LIN {X 0,Y 318.181,Z 414.797,A -85,B 0,C 180,E1 -16259.832,E2 -16259.832} C_VEL
LIN {X 0,Y 315.515,Z 502.273,A -85,B 0,C 180,E1 -16261.797,E2 -16261.797} C_VEL
LIN {X 0,Y 314.622,Z 517.231,A -85,B 0,C 180,E1 -16262.298,E2 -16262.298} C_VEL
LIN {X 0,Y 313.283,Z 530.709,A -85,B 0,C 180,E1 -16262.984,E2 -16262.984} C_VEL
LIN {X 0,Y 311.702,Z 543.956,A -85,B 0,C 180,E1 -16263.92,E2 -16263.92} C_VEL
LIN {X 0,Y 309.801,Z 557.279,A -85,B 0,C 180,E1 -16265.151,E2 -16265.151} C_VEL
LIN {X 0,Y 307.763,Z 569.737,A -85,B 0,C 180,E1 -16266.626,E2 -16266.626} C_VEL
LIN {X 0,Y 305.798,Z 579.793,A -85,B 0,C 180,E1 -16268.073,E2 -16268.073} C_VEL
LIN {X 0,Y 303.56,Z 590.854,A -85,B 0,C 180,E1 -16270.035,E2 -16270.035} C_VEL
LIN {X 0,Y 301.653,Z 599.979,A -85,B 0,C 180,E1 -16272.021,E2 -16272.021} C_VEL
LIN {X 0,Y 299.984,Z 608.705,A -85,B 0,C 180,E1 -16274.372,E2 -16274.372} C_VEL
LIN {X 0,Y 298.796,Z 614.845,A -85,B 0,C 180,E1 -16276.398,E2 -16276.398} C_VEL
LIN {X 0,Y 297.807,Z 619.932,A -85,B 0,C 180,E1 -16278.431,E2 -16278.431} C_VEL
LIN {X 0,Y 297.035,Z 625.187,A -85,B 0,C 180,E1 -16281.155,E2 -16281.155} C_VEL
LIN {X 0,Y 296.688,Z 628.133,A -85,B 0,C 180,E1 -16283.2,E2 -16283.2} C_VEL
LIN {X 0,Y 296.486,Z 630.822,A -85,B 0,C 180,E1 -16285.924,E2 -16285.924} C_VEL
LIN {X 0,Y 296.446,Z 632.15,A -85,B 0,C 180,E1 -16288.644,E2 -16288.644} C_VEL
LIN {X 0,Y 296.447,Z 632.143,A -85,B 0,C 180,E1 -16291.36,E2 -16291.36} C_VEL
LIN {X 0,Y 296.487,Z 630.798,A -85,B 0,C 180,E1 -16294.08,E2 -16294.08} C_VEL
LIN {X 0,Y 296.695,Z 628.094,A -85,B 0,C 180,E1 -16296.804,E2 -16296.804} C_VEL
LIN {X 0,Y 297.195,Z 623.958,A -85,B 0,C 180,E1 -16299.53,E2 -16299.53} C_VEL
LIN {X 0,Y 298.059,Z 618.26,A -85,B 0,C 180,E1 -16302.254,E2 -16302.254} C_VEL
LIN {X 0,Y 299.398,Z 611.836,A -85,B 0,C 180,E1 -16304.618,E2 -16304.618} C_VEL
LIN {X 0,Y 300.846,Z 603.858,A -85,B 0,C 180,E1 -16306.98,E2 -16306.98} C_VEL
LIN {X 0,Y 302.56,Z 595.508,A -85,B 0,C 180,E1 -16308.979,E2 -16308.979} C_VEL
LIN {X 0,Y 304.663,Z 585.459,A -85,B 0,C 180,E1 -16310.952,E2 -16310.952} C_VEL
LIN {X 0,Y 306.858,Z 574.243,A -85,B 0,C 180,E1 -16312.738,E2 -16312.738} C_VEL
LIN {X 0,Y 308.806,Z 563.08,A -85,B 0,C 180,E1 -16314.185,E2 -16314.185} C_VEL
LIN {X 0,Y 310.702,Z 550.92,A -85,B 0,C 180,E1 -16315.455,E2 -16315.455} C_VEL
LIN {X 0,Y 312.337,Z 538.56,A -85,B 0,C 180,E1 -16316.477,E2 -16316.477} C_VEL
LIN {X 0,Y 313.896,Z 524.825,A -85,B 0,C 180,E1 -16317.324,E2 -16317.324} C_VEL
LIN {X 0,Y 315.02,Z 510.572,A -85,B 0,C 180,E1 -16317.939,E2 -16317.939} C_VEL
LIN {X 0,Y 315.853,Z 497.641,A -85,B 0,C 180,E1 -16318.356,E2 -16318.356} C_VEL
LIN {X 0,Y 321.075,Z 453.072,A -85,B 0,C 180,E1 -16320.185,E2 -16320.185} C_VEL
LIN {X 0,Y 325.694,Z 416.284,A -85,B 0,C 180,E1 -16321.698,E2 -16321.698} C_VEL
LIN {X 0,Y 325.549,Z 408.176,A -85,B 0,C 180,E1 -16322.367,E2 -16322.367} C_VEL
LIN {X 0,Y 323.178,Z 401.098,A -85,B 0,C 180,E1 -16323.67,E2 -16323.67} C_VEL
LIN {X 0,Y 321.541,Z 396.245,A -85,B 0,C 180,E1 -16324.752,E2 -16324.752} C_VEL
LIN {X 0,Y 321.234,Z 394.789,A -85,B 0,C 180,E1 -16325.171,E2 -16325.171} C_VEL
LIN {X 0,Y 319.761,Z 392.123,A -85,B 0,C 180,E1 -16326.403,E2 -16326.403} C_VEL
LIN {X 0,Y 317.084,Z 387.927,A -85,B 0,C 180,E1 -16329.126,E2 -16329.126} C_VEL
LIN {X 0,Y 315.872,Z 386.212,A -85,B 0,C 180,E1 -16330.845,E2 -16330.845} C_VEL
LIN {X 0,Y 314.928,Z 385.265,A -85,B 0,C 180,E1 -16332.571,E2 -16332.571} C_VEL
LIN {X 0,Y 314.162,Z 384.822,A -85,B 0,C 180,E1 -16335.716,E2 -16335.716} C_VEL
LIN {X 0,Y 314.202,Z 385.504,A -85,B 0,C 180,E1 -16337.853,E2 -16337.853} C_VEL
LIN {X 0,Y 314.421,Z 386.794,A -85,B 0,C 180,E1 -16339.593,E2 -16339.593} C_VEL
LIN {X 0,Y 315.302,Z 390.269,A -85,B 0,C 180,E1 -16342.63,E2 -16342.63} C_VEL
LIN {X 0,Y 318.949,Z 396.314,A -85,B 0,C 180,E1 -16345.133,E2 -16345.133} C_VEL
LIN {X 0,Y 322.085,Z 401.94,A -85,B 0,C 180,E1 -16346.841,E2 -16346.841} C_VEL
LIN {X 0,Y 324.388,Z 406.46,A -85,B 0,C 180,E1 -16347.96,E2 -16347.96} C_VEL
LIN {X 0,Y 327.507,Z 413.311,A -85,B 0,C 180,E1 -16349.361,E2 -16349.361} C_VEL
LIN {X 0,Y 328.621,Z 416.471,A -85,B 0,C 180,E1 -16349.868,E2 -16349.868} C_VEL
LIN {X 0,Y 329.285,Z 421.801,A -85,B 0,C 180,E1 -16350.398,E2 -16350.398} C_VEL
LIN {X 0,Y 320.437,Z 500.804,A -85,B 0,C 180,E1 -16353.544,E2 -16353.544} C_VEL
LIN {X 0,Y 318.54,Z 515.101,A -85,B 0,C 180,E1 -16354.43,E2 -16354.43} C_VEL
LIN {X 0,Y 316.577,Z 526.868,A -85,B 0,C 180,E1 -16355.402,E2 -16355.402} C_VEL
LIN {X 0,Y 314.31,Z 538.512,A -85,B 0,C 180,E1 -16356.616,E2 -16356.616} C_VEL
LIN {X 0,Y 311.806,Z 549.386,A -85,B 0,C 180,E1 -16358.034,E2 -16358.034} C_VEL
LIN {X 0,Y 309.219,Z 559.762,A -85,B 0,C 180,E1 -16359.72,E2 -16359.72} C_VEL
LIN {X 0,Y 306.57,Z 569.095,A -85,B 0,C 180,E1 -16361.626,E2 -16361.626} C_VEL
LIN {X 0,Y 304.38,Z 576.647,A -85,B 0,C 180,E1 -16363.57,E2 -16363.57} C_VEL
LIN {X 0,Y 302.686,Z 581.817,A -85,B 0,C 180,E1 -16365.202,E2 -16365.202} C_VEL
LIN {X 0,Y 301.046,Z 586.845,A -85,B 0,C 180,E1 -16367.186,E2 -16367.186} C_VEL
LIN {X 0,Y 299.652,Z 590.71,A -85,B 0,C 180,E1 -16369.186,E2 -16369.186} C_VEL
LIN {X 0,Y 298.514,Z 593.752,A -85,B 0,C 180,E1 -16371.432,E2 -16371.432} C_VEL
LIN {X 0,Y 297.737,Z 595.31,A -85,B 0,C 180,E1 -16373.222,E2 -16373.222} C_VEL
LIN {X 0,Y 297.348,Z 595.96,A -85,B 0,C 180,E1 -16374.575,E2 -16374.575} C_VEL
LIN {X 0,Y 297.123,Z 596.176,A -85,B 0,C 180,E1 -16375.931,E2 -16375.931} C_VEL
LIN {X 0,Y 296.911,Z 595.987,A -85,B 0,C 180,E1 -16377.287,E2 -16377.287} C_VEL
LIN {X 0,Y 296.735,Z 595.36,A -85,B 0,C 180,E1 -16378.643,E2 -16378.643} C_VEL
LIN {X 0,Y 296.629,Z 594.272,A -85,B 0,C 180,E1 -16380,E2 -16380} C_VEL
LIN {X 0,Y 296.615,Z 592.763,A -85,B 0,C 180,E1 -16381.358,E2 -16381.358} C_VEL
LIN {X 0,Y 296.749,Z 589.624,A -85,B 0,C 180,E1 -16383.394,E2 -16383.394} C_VEL
LIN {X 0,Y 296.833,Z 585.354,A -85,B 0,C 180,E1 -16385.435,E2 -16385.435} C_VEL
LIN {X 0,Y 297.207,Z 578.751,A -85,B 0,C 180,E1 -16387.815,E2 -16387.815} C_VEL
LIN {X 0,Y 297.663,Z 571.555,A -85,B 0,C 180,E1 -16389.856,E2 -16389.856} C_VEL
LIN {X 0,Y 298.297,Z 562.517,A -85,B 0,C 180,E1 -16391.897,E2 -16391.897} C_VEL
LIN {X 0,Y 299.162,Z 552.289,A -85,B 0,C 180,E1 -16393.76,E2 -16393.76} C_VEL
LIN {X 0,Y 300.011,Z 541.96,A -85,B 0,C 180,E1 -16395.28,E2 -16395.28} C_VEL
LIN {X 0,Y 300.804,Z 530.328,A -85,B 0,C 180,E1 -16396.675,E2 -16396.675} C_VEL
LIN {X 0,Y 301.521,Z 518.247,A -85,B 0,C 180,E1 -16397.814,E2 -16397.814} C_VEL
LIN {X 0,Y 302.325,Z 505.7,A -85,B 0,C 180,E1 -16398.729,E2 -16398.729} C_VEL
LIN {X 0,Y 302.867,Z 492.085,A -85,B 0,C 180,E1 -16399.442,E2 -16399.442} C_VEL
LIN {X 0,Y 305.687,Z 408.397,A -85,B 0,C 180,E1 -16402.326,E2 -16402.326} C_VEL
LIN {X 0,Y 302.216,Z 381.764,A -85,B 0,C 180,E1 -16403.423,E2 -16403.423} C_VEL
LIN {X 0,Y 302.408,Z 377.134,A -85,B 0,C 180,E1 -16404.363,E2 -16404.363} C_VEL
LIN {X 0,Y 300.168,Z 364.932,A -85,B 0,C 180,E1 -16407.16,E2 -16407.16} C_VEL
LIN {X 0,Y 298.492,Z 356.928,A -85,B 0,C 180,E1 -16409.062,E2 -16409.062} C_VEL
LIN {X 0,Y 298.403,Z 356.939,A -85,B 0,C 180,E1 -16412.799,E2 -16412.799} C_VEL
LIN {X 0,Y 298.433,Z 356.935,A -85,B 0,C 180,E1 -16416.802,E2 -16416.802} C_VEL
LIN {X 0,Y 298.354,Z 356.945,A -85,B 0,C 180,E1 -16421.267,E2 -16421.267} C_VEL
LIN {X 0,Y 298.361,Z 356.945,A -85,B 0,C 180,E1 -16425.034,E2 -16425.034} C_VEL
LIN {X 0,Y 298.354,Z 356.946,A -85,B 0,C 180,E1 -16428.92,E2 -16428.92} C_VEL
LIN {X 0,Y 298.403,Z 356.941,A -85,B 0,C 180,E1 -16432.238,E2 -16432.238} C_VEL
LIN {X 0,Y 298.498,Z 357.128,A -85,B 0,C 180,E1 -16433.939,E2 -16433.939} C_VEL
LIN {X 0,Y 300.452,Z 364.93,A -85,B 0,C 180,E1 -16436.673,E2 -16436.673} C_VEL
LIN {X 0,Y 309.752,Z 383.967,A -85,B 0,C 180,E1 -16438.311,E2 -16438.311} C_VEL
LIN {X 0,Y 317.575,Z 402.728,A -85,B 0,C 180,E1 -16439.664,E2 -16439.664} C_VEL
LIN {X 0,Y 318.397,Z 408.082,A -85,B 0,C 180,E1 -16439.888,E2 -16439.888} C_VEL
LIN {X 0,Y 315.383,Z 501.879,A -85,B 0,C 180,E1 -16442.006,E2 -16442.006} C_VEL
LIN {X 0,Y 314.601,Z 514.095,A -85,B 0,C 180,E1 -16442.472,E2 -16442.472} C_VEL
LIN {X 0,Y 313.135,Z 528.181,A -85,B 0,C 180,E1 -16443.236,E2 -16443.236} C_VEL
LIN {X 0,Y 311.532,Z 541.631,A -85,B 0,C 180,E1 -16444.259,E2 -16444.259} C_VEL
LIN {X 0,Y 309.826,Z 553.788,A -85,B 0,C 180,E1 -16445.45,E2 -16445.45} C_VEL
LIN {X 0,Y 307.687,Z 566.235,A -85,B 0,C 180,E1 -16446.971,E2 -16446.971} C_VEL
LIN {X 0,Y 305.392,Z 577.917,A -85,B 0,C 180,E1 -16448.747,E2 -16448.747} C_VEL
LIN {X 0,Y 303.28,Z 588.352,A -85,B 0,C 180,E1 -16450.716,E2 -16450.716} C_VEL
LIN {X 0,Y 301.506,Z 596.934,A -85,B 0,C 180,E1 -16452.702,E2 -16452.702} C_VEL
LIN {X 0,Y 299.992,Z 605.205,A -85,B 0,C 180,E1 -16455.064,E2 -16455.064} C_VEL
LIN {X 0,Y 298.702,Z 610.956,A -85,B 0,C 180,E1 -16457.082,E2 -16457.082} C_VEL
LIN {X 0,Y 297.848,Z 615.682,A -85,B 0,C 180,E1 -16459.117,E2 -16459.117} C_VEL
LIN {X 0,Y 297.072,Z 620.571,A -85,B 0,C 180,E1 -16461.838,E2 -16461.838} C_VEL
LIN {X 0,Y 296.69,Z 623.976,A -85,B 0,C 180,E1 -16464.561,E2 -16464.561} C_VEL
LIN {X 0,Y 296.541,Z 626,A -85,B 0,C 180,E1 -16467.281,E2 -16467.281} C_VEL
LIN {X 0,Y 296.452,Z 626.694,A -85,B 0,C 180,E1 -16469.998,E2 -16469.998} C_VEL
LIN {X 0,Y 296.539,Z 626.066,A -85,B 0,C 180,E1 -16472.715,E2 -16472.715} C_VEL
LIN {X 0,Y 296.668,Z 624.104,A -85,B 0,C 180,E1 -16475.435,E2 -16475.435} C_VEL
LIN {X 0,Y 297.056,Z 620.755,A -85,B 0,C 180,E1 -16478.159,E2 -16478.159} C_VEL
LIN {X 0,Y 297.809,Z 615.922,A -85,B 0,C 180,E1 -16480.88,E2 -16480.88} C_VEL
LIN {X 0,Y 299.059,Z 609.457,A -85,B 0,C 180,E1 -16483.59,E2 -16483.59} C_VEL
LIN {X 0,Y 300.295,Z 603.371,A -85,B 0,C 180,E1 -16485.611,E2 -16485.611} C_VEL
LIN {X 0,Y 301.715,Z 596.064,A -85,B 0,C 180,E1 -16487.624,E2 -16487.624} C_VEL
LIN {X 0,Y 303.553,Z 587.276,A -85,B 0,C 180,E1 -16489.613,E2 -16489.613} C_VEL
LIN {X 0,Y 305.738,Z 576.623,A -85,B 0,C 180,E1 -16491.577,E2 -16491.577} C_VEL
LIN {X 0,Y 307.797,Z 565.849,A -85,B 0,C 180,E1 -16493.193,E2 -16493.193} C_VEL
LIN {X 0,Y 309.792,Z 554.196,A -85,B 0,C 180,E1 -16494.617,E2 -16494.617} C_VEL
LIN {X 0,Y 311.623,Z 541.043,A -85,B 0,C 180,E1 -16495.908,E2 -16495.908} C_VEL
LIN {X 0,Y 313.318,Z 527.366,A -85,B 0,C 180,E1 -16496.922,E2 -16496.922} C_VEL
LIN {X 0,Y 314.674,Z 512.864,A -85,B 0,C 180,E1 -16497.697,E2 -16497.697} C_VEL
LIN {X 0,Y 315.593,Z 498.5,A -85,B 0,C 180,E1 -16498.196,E2 -16498.196} C_VEL
LIN {X 0,Y 318.051,Z 420.026,A -85,B 0,C 180,E1 -16499.96,E2 -16499.96} C_VEL
LIN {X 0,Y 317.598,Z 416.226,A -85,B 0,C 180,E1 -16500.104,E2 -16500.104} C_VEL
LIN {X 0,Y 316.27,Z 412.711,A -85,B 0,C 180,E1 -16500.335,E2 -16500.335} C_VEL
LIN {X 0,Y 310.742,Z 402.776,A -85,B 0,C 180,E1 -16501.197,E2 -16501.197} C_VEL
LIN {X 0,Y 310.267,Z 401.571,A -85,B 0,C 180,E1 -16501.282,E2 -16501.282} C_VEL
LIN {X 0,Y 303.441,Z 385.758,A -85,B 0,C 180,E1 -16502.503,E2 -16502.503} C_VEL
LIN {X 0,Y 296.623,Z 371.72,A -85,B 0,C 180,E1 -16503.748,E2 -16503.748} C_VEL
LIN {X 0,Y 293.184,Z 364.851,A -85,B 0,C 180,E1 -16504.427,E2 -16504.427} C_VEL
LIN {X 0,Y 291.391,Z 357.815,A -85,B 0,C 180,E1 -16507.08,E2 -16507.08} C_VEL
LIN {X 0,Y 291.286,Z 357.826,A -85,B 0,C 180,E1 -16511.586,E2 -16511.586} C_VEL
LIN {X 0,Y 291.273,Z 357.827,A -85,B 0,C 180,E1 -16515.594,E2 -16515.594} C_VEL
LIN {X 0,Y 291.29,Z 357.827,A -85,B 0,C 180,E1 -16519.35,E2 -16519.35} C_VEL
LIN {X 0,Y 291.375,Z 357.804,A -85,B 0,C 180,E1 -16522.915,E2 -16522.915} C_VEL
LIN {X 0,Y 291.332,Z 357.807,A -85,B 0,C 180,E1 -16526.3,E2 -16526.3} C_VEL
LIN {X 0,Y 291.352,Z 357.818,A -85,B 0,C 180,E1 -16530.267,E2 -16530.267} C_VEL
LIN {X 0,Y 291.345,Z 357.796,A -85,B 0,C 180,E1 -16534.265,E2 -16534.265} C_VEL
LIN {X 0,Y 291.351,Z 357.817,A -85,B 0,C 180,E1 -16537.297,E2 -16537.297} C_VEL
LIN {X 0,Y 291.379,Z 357.788,A -85,B 0,C 180,E1 -16540.264,E2 -16540.264} C_VEL
LIN {X 0,Y 291.485,Z 357.804,A -85,B 0,C 180,E1 -16544.664,E2 -16544.664} C_VEL
LIN {X 0,Y 291.515,Z 357.799,A -85,B 0,C 180,E1 -16548.88,E2 -16548.88} C_VEL
LIN {X 0,Y 291.636,Z 357.777,A -85,B 0,C 180,E1 -16551.686,E2 -16551.686} C_VEL
LIN {X 0,Y 291.584,Z 357.785,A -85,B 0,C 180,E1 -16554.467,E2 -16554.467} C_VEL
LIN {X 0,Y 291.857,Z 357.752,A -85,B 0,C 180,E1 -16558.62,E2 -16558.62} C_VEL
LIN {X 0,Y 291.866,Z 357.753,A -85,B 0,C 180,E1 -16561.38,E2 -16561.38} C_VEL
LIN {X 0,Y 291.673,Z 357.777,A -85,B 0,C 180,E1 -16566.92,E2 -16566.92} C_VEL
LIN {X 0,Y 291.554,Z 357.789,A -85,B 0,C 180,E1 -16569.714,E2 -16569.714} C_VEL
LIN {X 0,Y 291.501,Z 357.795,A -85,B 0,C 180,E1 -16573.951,E2 -16573.951} C_VEL
LIN {X 0,Y 291.417,Z 357.803,A -85,B 0,C 180,E1 -16576.822,E2 -16576.822} C_VEL
LIN {X 0,Y 291.378,Z 357.812,A -85,B 0,C 180,E1 -16579.843,E2 -16579.843} C_VEL
LIN {X 0,Y 291.313,Z 357.812,A -85,B 0,C 180,E1 -16584.213,E2 -16584.213} C_VEL
LIN {X 0,Y 291.316,Z 357.816,A -85,B 0,C 180,E1 -16587.282,E2 -16587.282} C_VEL
LIN {X 0,Y 291.289,Z 357.815,A -85,B 0,C 180,E1 -16590.442,E2 -16590.442} C_VEL
LIN {X 0,Y 291.332,Z 357.816,A -85,B 0,C 180,E1 -16593.7,E2 -16593.7} C_VEL
LIN {X 0,Y 291.341,Z 357.82,A -85,B 0,C 180,E1 -16597.249,E2 -16597.249} C_VEL
LIN {X 0,Y 291.288,Z 357.824,A -85,B 0,C 180,E1 -16600.65,E2 -16600.65} C_VEL
LIN {X 0,Y 291.272,Z 357.831,A -85,B 0,C 180,E1 -16604.405,E2 -16604.405} C_VEL
LIN {X 0,Y 291.285,Z 357.83,A -85,B 0,C 180,E1 -16608.413,E2 -16608.413} C_VEL
LIN {X 0,Y 291.364,Z 357.957,A -85,B 0,C 180,E1 -16611.73,E2 -16611.73} C_VEL
LIN {X 0,Y 293.787,Z 366.948,A -85,B 0,C 180,E1 -16614.964,E2 -16614.964} C_VEL
LIN {X 0,Y 294.381,Z 369.415,A -85,B 0,C 180,E1 -16615.805,E2 -16615.805} C_VEL
LIN {X 0,Y 303.664,Z 388.91,A -85,B 0,C 180,E1 -16617.522,E2 -16617.522} C_VEL
LIN {X 0,Y 309.907,Z 403.802,A -85,B 0,C 180,E1 -16618.649,E2 -16618.649} C_VEL
LIN {X 0,Y 312.081,Z 416.22,A -85,B 0,C 180,E1 -16619.217,E2 -16619.217} C_VEL
LIN {X 0,Y 309.113,Z 506.688,A -85,B 0,C 180,E1 -16621.298,E2 -16621.298} C_VEL
LIN {X 0,Y 308.029,Z 520.691,A -85,B 0,C 180,E1 -16621.838,E2 -16621.838} C_VEL
LIN {X 0,Y 306.571,Z 534.345,A -85,B 0,C 180,E1 -16622.62,E2 -16622.62} C_VEL
LIN {X 0,Y 304.792,Z 547.616,A -85,B 0,C 180,E1 -16623.651,E2 -16623.651} C_VEL
LIN {X 0,Y 302.863,Z 560.156,A -85,B 0,C 180,E1 -16624.916,E2 -16624.916} C_VEL
LIN {X 0,Y 300.81,Z 572.022,A -85,B 0,C 180,E1 -16626.418,E2 -16626.418} C_VEL
LIN {X 0,Y 298.742,Z 581.694,A -85,B 0,C 180,E1 -16627.891,E2 -16627.891} C_VEL
LIN {X 0,Y 296.499,Z 592.417,A -85,B 0,C 180,E1 -16629.9,E2 -16629.9} C_VEL
LIN {X 0,Y 294.563,Z 601.27,A -85,B 0,C 180,E1 -16631.933,E2 -16631.933} C_VEL
LIN {X 0,Y 292.871,Z 609.756,A -85,B 0,C 180,E1 -16634.34,E2 -16634.34} C_VEL
LIN {X 0,Y 291.477,Z 616.591,A -85,B 0,C 180,E1 -16636.761,E2 -16636.761} C_VEL
LIN {X 0,Y 290.577,Z 621.302,A -85,B 0,C 180,E1 -16638.846,E2 -16638.846} C_VEL
LIN {X 0,Y 289.846,Z 626.189,A -85,B 0,C 180,E1 -16641.637,E2 -16641.637} C_VEL
LIN {X 0,Y 289.471,Z 629.68,A -85,B 0,C 180,E1 -16644.521,E2 -16644.521} C_VEL
LIN {X 0,Y 289.388,Z 631.588,A -85,B 0,C 180,E1 -16647.218,E2 -16647.218} C_VEL
LIN {X 0,Y 289.37,Z 632.246,A -85,B 0,C 180,E1 -16650.002,E2 -16650.002} C_VEL
LIN {X 0,Y 289.389,Z 631.571,A -85,B 0,C 180,E1 -16652.786,E2 -16652.786} C_VEL
LIN {X 0,Y 289.481,Z 629.551,A -85,B 0,C 180,E1 -16655.575,E2 -16655.575} C_VEL
LIN {X 0,Y 289.861,Z 626.143,A -85,B 0,C 180,E1 -16658.367,E2 -16658.367} C_VEL
LIN {X 0,Y 290.58,Z 621.246,A -85,B 0,C 180,E1 -16661.158,E2 -16661.158} C_VEL
LIN {X 0,Y 291.481,Z 616.519,A -85,B 0,C 180,E1 -16663.244,E2 -16663.244} C_VEL
LIN {X 0,Y 292.868,Z 609.664,A -85,B 0,C 180,E1 -16665.664,E2 -16665.664} C_VEL
LIN {X 0,Y 294.566,Z 601.158,A -85,B 0,C 180,E1 -16668.071,E2 -16668.071} C_VEL
LIN {X 0,Y 296.502,Z 592.281,A -85,B 0,C 180,E1 -16670.104,E2 -16670.104} C_VEL
LIN {X 0,Y 298.747,Z 581.531,A -85,B 0,C 180,E1 -16672.113,E2 -16672.113} C_VEL
LIN {X 0,Y 300.989,Z 570.65,A -85,B 0,C 180,E1 -16673.754,E2 -16673.754} C_VEL
LIN {X 0,Y 303.132,Z 558.555,A -85,B 0,C 180,E1 -16675.241,E2 -16675.241} C_VEL
LIN {X 0,Y 305.032,Z 545.501,A -85,B 0,C 180,E1 -16676.515,E2 -16676.515} C_VEL
LIN {X 0,Y 307.888,Z 525.854,A -85,B 0,C 180,E1 -16677.995,E2 -16677.995} C_VEL
LIN {X 0,Y 309.583,Z 512.084,A -85,B 0,C 180,E1 -16678.752,E2 -16678.752} C_VEL
LIN {X 0,Y 316.684,Z 455.092,A -85,B 0,C 180,E1 -16681.141,E2 -16681.141} C_VEL
LIN {X 0,Y 321.69,Z 418.334,A -85,B 0,C 180,E1 -16682.669,E2 -16682.669} C_VEL
LIN {X 0,Y 321.657,Z 412.005,A -85,B 0,C 180,E1 -16683.213,E2 -16683.213} C_VEL
LIN {X 0,Y 319.912,Z 406.208,A -85,B 0,C 180,E1 -16684.323,E2 -16684.323} C_VEL
LIN {X 0,Y 317.902,Z 400.512,A -85,B 0,C 180,E1 -16685.657,E2 -16685.657} C_VEL
LIN {X 0,Y 314.755,Z 396.173,A -85,B 0,C 180,E1 -16687.662,E2 -16687.662} C_VEL
LIN {X 0,Y 313.481,Z 394.308,A -85,B 0,C 180,E1 -16688.885,E2 -16688.885} C_VEL
LIN {X 0,Y 312.065,Z 392.237,A -85,B 0,C 180,E1 -16690.778,E2 -16690.778} C_VEL
LIN {X 0,Y 310.582,Z 390.824,A -85,B 0,C 180,E1 -16693.605,E2 -16693.605} C_VEL
LIN {X 0,Y 310.017,Z 390.757,A -85,B 0,C 180,E1 -16696.507,E2 -16696.507} C_VEL
LIN {X 0,Y 310.122,Z 392.046,A -85,B 0,C 180,E1 -16698.913,E2 -16698.913} C_VEL
LIN {X 0,Y 312.611,Z 396.096,A -85,B 0,C 180,E1 -16701.895,E2 -16701.895} C_VEL
LIN {X 0,Y 315.852,Z 401.54,A -85,B 0,C 180,E1 -16704.393,E2 -16704.393} C_VEL
LIN {X 0,Y 318.844,Z 407.285,A -85,B 0,C 180,E1 -16706.215,E2 -16706.215} C_VEL
LIN {X 0,Y 321.387,Z 412.56,A -85,B 0,C 180,E1 -16707.564,E2 -16707.564} C_VEL
LIN {X 0,Y 324.493,Z 419.929,A -85,B 0,C 180,E1 -16709.054,E2 -16709.054} C_VEL
LIN {X 0,Y 324.888,Z 423.919,A -85,B 0,C 180,E1 -16709.461,E2 -16709.461} C_VEL
LIN {X 0,Y 315.587,Z 501.078,A -85,B 0,C 180,E1 -16712.612,E2 -16712.612} C_VEL
LIN {X 0,Y 313.452,Z 515.756,A -85,B 0,C 180,E1 -16713.537,E2 -16713.537} C_VEL
LIN {X 0,Y 311.208,Z 528.176,A -85,B 0,C 180,E1 -16714.591,E2 -16714.591} C_VEL
LIN {X 0,Y 308.499,Z 540.821,A -85,B 0,C 180,E1 -16715.97,E2 -16715.97} C_VEL
LIN {X 0,Y 305.659,Z 552.109,A -85,B 0,C 180,E1 -16717.526,E2 -16717.526} C_VEL
LIN {X 0,Y 302.852,Z 562.164,A -85,B 0,C 180,E1 -16719.275,E2 -16719.275} C_VEL
LIN {X 0,Y 300.086,Z 571.129,A -85,B 0,C 180,E1 -16721.215,E2 -16721.215} C_VEL
LIN {X 0,Y 297.374,Z 579.378,A -85,B 0,C 180,E1 -16723.525,E2 -16723.525} C_VEL
LIN {X 0,Y 295.382,Z 584.987,A -85,B 0,C 180,E1 -16725.533,E2 -16725.533} C_VEL
LIN {X 0,Y 293.64,Z 589.407,A -85,B 0,C 180,E1 -16727.561,E2 -16727.561} C_VEL
LIN {X 0,Y 292.753,Z 591.686,A -85,B 0,C 180,E1 -16728.927,E2 -16728.927} C_VEL
LIN {X 0,Y 291.484,Z 594.625,A -85,B 0,C 180,E1 -16731.332,E2 -16731.332} C_VEL
LIN {X 0,Y 290.734,Z 595.92,A -85,B 0,C 180,E1 -16733.058,E2 -16733.058} C_VEL
LIN {X 0,Y 290.311,Z 596.458,A -85,B 0,C 180,E1 -16734.443,E2 -16734.443} C_VEL
LIN {X 0,Y 290.056,Z 596.585,A -85,B 0,C 180,E1 -16735.832,E2 -16735.832} C_VEL
LIN {X 0,Y 289.832,Z 596.275,A -85,B 0,C 180,E1 -16737.22,E2 -16737.22} C_VEL
LIN {X 0,Y 289.65,Z 595.513,A -85,B 0,C 180,E1 -16738.61,E2 -16738.61} C_VEL
LIN {X 0,Y 289.543,Z 594.338,A -85,B 0,C 180,E1 -16740,E2 -16740} C_VEL
LIN {X 0,Y 289.553,Z 591.724,A -85,B 0,C 180,E1 -16742.087,E2 -16742.087} C_VEL
LIN {X 0,Y 289.698,Z 588.036,A -85,B 0,C 180,E1 -16744.174,E2 -16744.174} C_VEL
LIN {X 0,Y 289.894,Z 582.403,A -85,B 0,C 180,E1 -16746.542,E2 -16746.542} C_VEL
LIN {X 0,Y 290.264,Z 575.769,A -85,B 0,C 180,E1 -16748.704,E2 -16748.704} C_VEL
LIN {X 0,Y 290.836,Z 567.725,A -85,B 0,C 180,E1 -16750.794,E2 -16750.794} C_VEL
LIN {X 0,Y 291.601,Z 557.661,A -85,B 0,C 180,E1 -16752.882,E2 -16752.882} C_VEL
LIN {X 0,Y 292.369,Z 548.439,A -85,B 0,C 180,E1 -16754.442,E2 -16754.442} C_VEL
LIN {X 0,Y 293.255,Z 537.159,A -85,B 0,C 180,E1 -16755.998,E2 -16755.998} C_VEL
LIN {X 0,Y 294.14,Z 524.634,A -85,B 0,C 180,E1 -16757.377,E2 -16757.377} C_VEL
LIN {X 0,Y 294.943,Z 511.46,A -85,B 0,C 180,E1 -16758.495,E2 -16758.495} C_VEL
LIN {X 0,Y 295.618,Z 497.641,A -85,B 0,C 180,E1 -16759.351,E2 -16759.351} C_VEL
LIN {X 0,Y 296.256,Z 482.294,A -85,B 0,C 180,E1 -16759.984,E2 -16759.984} C_VEL
LIN {X 0,Y 298.73,Z 409.096,A -85,B 0,C 180,E1 -16762.579,E2 -16762.579} C_VEL
LIN {X 0,Y 295.229,Z 381.64,A -85,B 0,C 180,E1 -16763.758,E2 -16763.758} C_VEL
LIN {X 0,Y 295.389,Z 377.94,A -85,B 0,C 180,E1 -16764.56,E2 -16764.56} C_VEL
LIN {X 0,Y 292.812,Z 364.332,A -85,B 0,C 180,E1 -16767.729,E2 -16767.729} C_VEL
LIN {X 0,Y 291.455,Z 357.805,A -85,B 0,C 180,E1 -16769.286,E2 -16769.286} C_VEL
LIN {X 0,Y 291.352,Z 357.816,A -85,B 0,C 180,E1 -16773.698,E2 -16773.698} C_VEL
LIN {X 0,Y 291.359,Z 357.817,A -85,B 0,C 180,E1 -16777.247,E2 -16777.247} C_VEL
LIN {X 0,Y 291.301,Z 357.825,A -85,B 0,C 180,E1 -16781.588,E2 -16781.588} C_VEL
LIN {X 0,Y 291.288,Z 357.828,A -85,B 0,C 180,E1 -16785.595,E2 -16785.595} C_VEL
LIN {X 0,Y 291.306,Z 357.826,A -85,B 0,C 180,E1 -16789.351,E2 -16789.351} C_VEL
LIN {X 0,Y 291.408,Z 357.852,A -85,B 0,C 180,E1 -16793.134,E2 -16793.134} C_VEL
LIN {X 0,Y 293.312,Z 365.196,A -85,B 0,C 180,E1 -16795.755,E2 -16795.755} C_VEL
LIN {X 0,Y 302.995,Z 384.698,A -85,B 0,C 180,E1 -16797.536,E2 -16797.536} C_VEL
LIN {X 0,Y 310.198,Z 401.425,A -85,B 0,C 180,E1 -16798.826,E2 -16798.826} C_VEL
LIN {X 0,Y 311.886,Z 406.121,A -85,B 0,C 180,E1 -16799.138,E2 -16799.138} C_VEL
LIN {X 0,Y 312.27,Z 408.498,A -85,B 0,C 180,E1 -16799.242,E2 -16799.242} C_VEL
LIN {X 0,Y 309.149,Z 501.962,A -85,B 0,C 180,E1 -16801.39,E2 -16801.39} C_VEL
LIN {X 0,Y 308.315,Z 514.175,A -85,B 0,C 180,E1 -16801.862,E2 -16801.862} C_VEL
LIN {X 0,Y 306.818,Z 528.256,A -85,B 0,C 180,E1 -16802.64,E2 -16802.64} C_VEL
LIN {X 0,Y 305.15,Z 541.704,A -85,B 0,C 180,E1 -16803.68,E2 -16803.68} C_VEL
LIN {X 0,Y 303.309,Z 554.271,A -85,B 0,C 180,E1 -16804.939,E2 -16804.939} C_VEL
LIN {X 0,Y 301.154,Z 566.307,A -85,B 0,C 180,E1 -16806.442,E2 -16806.442} C_VEL
LIN {X 0,Y 298.769,Z 577.988,A -85,B 0,C 180,E1 -16808.252,E2 -16808.252} C_VEL
LIN {X 0,Y 296.576,Z 588.423,A -85,B 0,C 180,E1 -16810.262,E2 -16810.262} C_VEL
LIN {X 0,Y 294.642,Z 597.296,A -85,B 0,C 180,E1 -16812.364,E2 -16812.364} C_VEL
LIN {X 0,Y 293.101,Z 605.274,A -85,B 0,C 180,E1 -16814.705,E2 -16814.705} C_VEL
LIN {X 0,Y 291.75,Z 611.026,A -85,B 0,C 180,E1 -16816.769,E2 -16816.769} C_VEL
LIN {X 0,Y 290.843,Z 615.751,A -85,B 0,C 180,E1 -16818.852,E2 -16818.852} C_VEL
LIN {X 0,Y 290.019,Z 620.64,A -85,B 0,C 180,E1 -16821.638,E2 -16821.638} C_VEL
LIN {X 0,Y 289.606,Z 624.044,A -85,B 0,C 180,E1 -16824.428,E2 -16824.428} C_VEL
LIN {X 0,Y 289.448,Z 626.067,A -85,B 0,C 180,E1 -16827.214,E2 -16827.214} C_VEL
LIN {X 0,Y 289.373,Z 626.761,A -85,B 0,C 180,E1 -16829.998,E2 -16829.998} C_VEL
LIN {X 0,Y 289.446,Z 626.133,A -85,B 0,C 180,E1 -16832.781,E2 -16832.781} C_VEL
LIN {X 0,Y 289.604,Z 624.17,A -85,B 0,C 180,E1 -16835.568,E2 -16835.568} C_VEL
LIN {X 0,Y 290.007,Z 620.822,A -85,B 0,C 180,E1 -16838.358,E2 -16838.358} C_VEL
LIN {X 0,Y 290.81,Z 615.988,A -85,B 0,C 180,E1 -16841.145,E2 -16841.145} C_VEL
LIN {X 0,Y 291.722,Z 611.327,A -85,B 0,C 180,E1 -16843.228,E2 -16843.228} C_VEL
LIN {X 0,Y 293.243,Z 604.55,A -85,B 0,C 180,E1 -16845.639,E2 -16845.639} C_VEL
LIN {X 0,Y 294.636,Z 597.524,A -85,B 0,C 180,E1 -16847.691,E2 -16847.691} C_VEL
LIN {X 0,Y 296.507,Z 588.96,A -85,B 0,C 180,E1 -16849.738,E2 -16849.738} C_VEL
LIN {X 0,Y 298.732,Z 578.635,A -85,B 0,C 180,E1 -16851.746,E2 -16851.746} C_VEL
LIN {X 0,Y 301.047,Z 567.084,A -85,B 0,C 180,E1 -16853.562,E2 -16853.562} C_VEL
LIN {X 0,Y 303.129,Z 555.768,A -85,B 0,C 180,E1 -16855.001,E2 -16855.001} C_VEL
LIN {X 0,Y 304.782,Z 544.635,A -85,B 0,C 180,E1 -16856.166,E2 -16856.166} C_VEL
LIN {X 0,Y 306.453,Z 531.993,A -85,B 0,C 180,E1 -16857.206,E2 -16857.206} C_VEL
LIN {X 0,Y 307.963,Z 517.806,A -85,B 0,C 180,E1 -16858.076,E2 -16858.076} C_VEL
LIN {X 0,Y 309.064,Z 503.825,A -85,B 0,C 180,E1 -16858.661,E2 -16858.661} C_VEL
LIN {X 0,Y 310.047,Z 479.535,A -85,B 0,C 180,E1 -16859.257,E2 -16859.257} C_VEL
LIN {X 0,Y 312.254,Z 407.787,A -85,B 0,C 180,E1 -16860.897,E2 -16860.897} C_VEL
LIN {X 0,Y 311.265,Z 404.16,A -85,B 0,C 180,E1 -16861.102,E2 -16861.102} C_VEL
LIN {X 0,Y 310.267,Z 401.571,A -85,B 0,C 180,E1 -16861.282,E2 -16861.282} C_VEL
LIN {X 0,Y 307.751,Z 396.737,A -85,B 0,C 180,E1 -16861.697,E2 -16861.697} C_VEL
LIN {X 0,Y 304.401,Z 392.617,A -85,B 0,C 180,E1 -16862.2,E2 -16862.2} C_VEL
LIN {X 0,Y 295.996,Z 383.65,A -85,B 0,C 180,E1 -16863.488,E2 -16863.488} C_VEL
LIN {X 0,Y 293.178,Z 379.055,A -85,B 0,C 180,E1 -16863.987,E2 -16863.987} C_VEL
LIN {X 0,Y 285.997,Z 364.972,A -85,B 0,C 180,E1 -16865.406,E2 -16865.406} C_VEL
LIN {X 0,Y 284.29,Z 358.698,A -85,B 0,C 180,E1 -16867.879,E2 -16867.879} C_VEL
LIN {X 0,Y 284.228,Z 358.704,A -85,B 0,C 180,E1 -16872.115,E2 -16872.115} C_VEL
LIN {X 0,Y 284.229,Z 358.704,A -85,B 0,C 180,E1 -16876.184,E2 -16876.184} C_VEL
LIN {X 0,Y 284.273,Z 358.7,A -85,B 0,C 180,E1 -16880.028,E2 -16880.028} C_VEL
LIN {X 0,Y 284.308,Z 358.692,A -85,B 0,C 180,E1 -16883.61,E2 -16883.61} C_VEL
LIN {X 0,Y 284.295,Z 358.677,A -85,B 0,C 180,E1 -16887.189,E2 -16887.189} C_VEL
LIN {X 0,Y 284.324,Z 358.694,A -85,B 0,C 180,E1 -16890.372,E2 -16890.372} C_VEL
LIN {X 0,Y 284.292,Z 358.671,A -85,B 0,C 180,E1 -16893.578,E2 -16893.578} C_VEL
LIN {X 0,Y 284.314,Z 358.695,A -85,B 0,C 180,E1 -16896.702,E2 -16896.702} C_VEL
LIN {X 0,Y 284.319,Z 358.666,A -85,B 0,C 180,E1 -16901.256,E2 -16901.256} C_VEL
LIN {X 0,Y 284.449,Z 358.675,A -85,B 0,C 180,E1 -16905.695,E2 -16905.695} C_VEL
LIN {X 0,Y 284.5,Z 358.669,A -85,B 0,C 180,E1 -16910.042,E2 -16910.042} C_VEL
LIN {X 0,Y 284.626,Z 358.657,A -85,B 0,C 180,E1 -16912.908,E2 -16912.908} C_VEL
LIN {X 0,Y 284.824,Z 358.628,A -85,B 0,C 180,E1 -16918.586,E2 -16918.586} C_VEL
LIN {X 0,Y 284.832,Z 358.629,A -85,B 0,C 180,E1 -16921.414,E2 -16921.414} C_VEL
LIN {X 0,Y 284.628,Z 358.653,A -85,B 0,C 180,E1 -16927.092,E2 -16927.092} C_VEL
LIN {X 0,Y 284.5,Z 358.669,A -85,B 0,C 180,E1 -16929.958,E2 -16929.958} C_VEL
LIN {X 0,Y 284.449,Z 358.676,A -85,B 0,C 180,E1 -16934.304,E2 -16934.304} C_VEL
LIN {X 0,Y 284.32,Z 358.694,A -85,B 0,C 180,E1 -16938.744,E2 -16938.744} C_VEL
LIN {X 0,Y 284.294,Z 358.676,A -85,B 0,C 180,E1 -16943.299,E2 -16943.299} C_VEL
LIN {X 0,Y 284.273,Z 358.694,A -85,B 0,C 180,E1 -16947.131,E2 -16947.131} C_VEL
LIN {X 0,Y 284.261,Z 358.687,A -85,B 0,C 180,E1 -16950.085,E2 -16950.085} C_VEL
LIN {X 0,Y 284.293,Z 358.693,A -85,B 0,C 180,E1 -16952.947,E2 -16952.947} C_VEL
LIN {X 0,Y 284.306,Z 358.694,A -85,B 0,C 180,E1 -16956.39,E2 -16956.39} C_VEL
LIN {X 0,Y 284.271,Z 358.702,A -85,B 0,C 180,E1 -16960.001,E2 -16960.001} C_VEL
LIN {X 0,Y 284.223,Z 358.707,A -85,B 0,C 180,E1 -16964.19,E2 -16964.19} C_VEL
LIN {X 0,Y 284.23,Z 358.709,A -85,B 0,C 180,E1 -16968.12,E2 -16968.12} C_VEL
LIN {X 0,Y 284.327,Z 358.839,A -85,B 0,C 180,E1 -16970.93,E2 -16970.93} C_VEL
LIN {X 0,Y 286.797,Z 368.082,A -85,B 0,C 180,E1 -16974.373,E2 -16974.373} C_VEL
LIN {X 0,Y 287.223,Z 369.574,A -85,B 0,C 180,E1 -16974.836,E2 -16974.836} C_VEL
LIN {X 0,Y 296.596,Z 388.69,A -85,B 0,C 180,E1 -16976.644,E2 -16976.644} C_VEL
LIN {X 0,Y 303.957,Z 405.993,A -85,B 0,C 180,E1 -16978.024,E2 -16978.024} C_VEL
LIN {X 0,Y 305.958,Z 417.321,A -85,B 0,C 180,E1 -16978.563,E2 -16978.563} C_VEL
LIN {X 0,Y 302.913,Z 506.636,A -85,B 0,C 180,E1 -16980.654,E2 -16980.654} C_VEL
LIN {X 0,Y 301.771,Z 520.632,A -85,B 0,C 180,E1 -16981.2,E2 -16981.2} C_VEL
LIN {X 0,Y 300.284,Z 534.284,A -85,B 0,C 180,E1 -16981.997,E2 -16981.997} C_VEL
LIN {X 0,Y 298.429,Z 547.554,A -85,B 0,C 180,E1 -16983.045,E2 -16983.045} C_VEL
LIN {X 0,Y 296.274,Z 560.983,A -85,B 0,C 180,E1 -16984.435,E2 -16984.435} C_VEL
LIN {X 0,Y 294.049,Z 573.132,A -85,B 0,C 180,E1 -16986.029,E2 -16986.029} C_VEL
LIN {X 0,Y 291.73,Z 583.583,A -85,B 0,C 180,E1 -16987.704,E2 -16987.704} C_VEL
LIN {X 0,Y 289.47,Z 593.981,A -85,B 0,C 180,E1 -16989.761,E2 -16989.761} C_VEL
LIN {X 0,Y 287.475,Z 602.56,A -85,B 0,C 180,E1 -16991.841,E2 -16991.841} C_VEL
LIN {X 0,Y 285.754,Z 610.774,A -85,B 0,C 180,E1 -16994.306,E2 -16994.306} C_VEL
LIN {X 0,Y 284.549,Z 616.525,A -85,B 0,C 180,E1 -16996.432,E2 -16996.432} C_VEL
LIN {X 0,Y 283.554,Z 621.235,A -85,B 0,C 180,E1 -16998.566,E2 -16998.566} C_VEL
LIN {X 0,Y 282.792,Z 626.122,A -85,B 0,C 180,E1 -17001.427,E2 -17001.427} C_VEL
LIN {X 0,Y 282.385,Z 629.517,A -85,B 0,C 180,E1 -17004.289,E2 -17004.289} C_VEL
LIN {X 0,Y 282.298,Z 631.521,A -85,B 0,C 180,E1 -17007.148,E2 -17007.148} C_VEL
LIN {X 0,Y 282.293,Z 632.179,A -85,B 0,C 180,E1 -17010.002,E2 -17010.002} C_VEL
LIN {X 0,Y 282.298,Z 631.503,A -85,B 0,C 180,E1 -17012.856,E2 -17012.856} C_VEL
LIN {X 0,Y 282.408,Z 629.483,A -85,B 0,C 180,E1 -17015.715,E2 -17015.715} C_VEL
LIN {X 0,Y 282.803,Z 626.075,A -85,B 0,C 180,E1 -17018.577,E2 -17018.577} C_VEL
LIN {X 0,Y 283.558,Z 621.177,A -85,B 0,C 180,E1 -17021.438,E2 -17021.438} C_VEL
LIN {X 0,Y 284.552,Z 616.45,A -85,B 0,C 180,E1 -17023.572,E2 -17023.572} C_VEL
LIN {X 0,Y 285.989,Z 609.685,A -85,B 0,C 180,E1 -17026.022,E2 -17026.022} C_VEL
LIN {X 0,Y 287.483,Z 602.444,A -85,B 0,C 180,E1 -17028.163,E2 -17028.163} C_VEL
LIN {X 0,Y 289.471,Z 593.841,A -85,B 0,C 180,E1 -17030.243,E2 -17030.243} C_VEL
LIN {X 0,Y 291.735,Z 583.413,A -85,B 0,C 180,E1 -17032.3,E2 -17032.3} C_VEL
LIN {X 0,Y 294.26,Z 571.784,A -85,B 0,C 180,E1 -17034.144,E2 -17034.144} C_VEL
LIN {X 0,Y 298.107,Z 552.979,A -85,B 0,C 180,E1 -17036.613,E2 -17036.613} C_VEL
LIN {X 0,Y 300.311,Z 542.26,A -85,B 0,C 180,E1 -17037.72,E2 -17037.72} C_VEL
LIN {X 0,Y 302.877,Z 527.859,A -85,B 0,C 180,E1 -17038.879,E2 -17038.879} C_VEL
LIN {X 0,Y 304.891,Z 513.756,A -85,B 0,C 180,E1 -17039.711,E2 -17039.711} C_VEL
LIN {X 0,Y 312.719,Z 455.538,A -85,B 0,C 180,E1 -17042.214,E2 -17042.214} C_VEL
LIN {X 0,Y 317.922,Z 419.724,A -85,B 0,C 180,E1 -17043.738,E2 -17043.738} C_VEL
LIN {X 0,Y 317.952,Z 415.898,A -85,B 0,C 180,E1 -17044.083,E2 -17044.083} C_VEL
LIN {X 0,Y 316.446,Z 410.532,A -85,B 0,C 180,E1 -17045.175,E2 -17045.175} C_VEL
LIN {X 0,Y 315.104,Z 406.404,A -85,B 0,C 180,E1 -17046.192,E2 -17046.192} C_VEL
LIN {X 0,Y 312.295,Z 402.41,A -85,B 0,C 180,E1 -17048.128,E2 -17048.128} C_VEL
LIN {X 0,Y 309.777,Z 399.218,A -85,B 0,C 180,E1 -17050.444,E2 -17050.444} C_VEL
LIN {X 0,Y 308.215,Z 397.691,A -85,B 0,C 180,E1 -17052.611,E2 -17052.611} C_VEL
LIN {X 0,Y 307.427,Z 397.195,A -85,B 0,C 180,E1 -17055.13,E2 -17055.13} C_VEL
LIN {X 0,Y 307.754,Z 397.917,A -85,B 0,C 180,E1 -17057.531,E2 -17057.531} C_VEL
LIN {X 0,Y 308.659,Z 399.579,A -85,B 0,C 180,E1 -17059.415,E2 -17059.415} C_VEL
LIN {X 0,Y 311.016,Z 403.602,A -85,B 0,C 180,E1 -17062.119,E2 -17062.119} C_VEL
LIN {X 0,Y 313.822,Z 408.862,A -85,B 0,C 180,E1 -17064.351,E2 -17064.351} C_VEL
LIN {X 0,Y 316.37,Z 414.034,A -85,B 0,C 180,E1 -17065.973,E2 -17065.973} C_VEL
LIN {X 0,Y 318.984,Z 420.011,A -85,B 0,C 180,E1 -17067.447,E2 -17067.447} C_VEL
LIN {X 0,Y 320.653,Z 424.564,A -85,B 0,C 180,E1 -17068.344,E2 -17068.344} C_VEL
LIN {X 0,Y 320.633,Z 426.569,A -85,B 0,C 180,E1 -17068.504,E2 -17068.504} C_VEL
LIN {X 0,Y 310.865,Z 501.845,A -85,B 0,C 180,E1 -17071.656,E2 -17071.656} C_VEL
LIN {X 0,Y 308.673,Z 515.78,A -85,B 0,C 180,E1 -17072.544,E2 -17072.544} C_VEL
LIN {X 0,Y 306.275,Z 528.178,A -85,B 0,C 180,E1 -17073.602,E2 -17073.602} C_VEL
LIN {X 0,Y 303.459,Z 540.564,A -85,B 0,C 180,E1 -17074.961,E2 -17074.961} C_VEL
LIN {X 0,Y 300.338,Z 552.106,A -85,B 0,C 180,E1 -17076.559,E2 -17076.559} C_VEL
LIN {X 0,Y 297.576,Z 561.391,A -85,B 0,C 180,E1 -17078.163,E2 -17078.163} C_VEL
LIN {X 0,Y 294.584,Z 570.483,A -85,B 0,C 180,E1 -17080.125,E2 -17080.125} C_VEL
LIN {X 0,Y 292.361,Z 576.741,A -85,B 0,C 180,E1 -17081.79,E2 -17081.79} C_VEL
LIN {X 0,Y 290.005,Z 582.96,A -85,B 0,C 180,E1 -17083.818,E2 -17083.818} C_VEL
LIN {X 0,Y 288.045,Z 587.887,A -85,B 0,C 180,E1 -17085.878,E2 -17085.878} C_VEL
LIN {X 0,Y 286.279,Z 591.688,A -85,B 0,C 180,E1 -17087.956,E2 -17087.956} C_VEL
LIN {X 0,Y 285.146,Z 594.405,A -85,B 0,C 180,E1 -17090.065,E2 -17090.065} C_VEL
LIN {X 0,Y 284.36,Z 595.67,A -85,B 0,C 180,E1 -17091.472,E2 -17091.472} C_VEL
LIN {X 0,Y 283.735,Z 596.521,A -85,B 0,C 180,E1 -17092.886,E2 -17092.886} C_VEL
LIN {X 0,Y 283.277,Z 596.963,A -85,B 0,C 180,E1 -17094.305,E2 -17094.305} C_VEL
LIN {X 0,Y 282.994,Z 596.952,A -85,B 0,C 180,E1 -17095.727,E2 -17095.727} C_VEL
LIN {X 0,Y 282.756,Z 596.506,A -85,B 0,C 180,E1 -17097.151,E2 -17097.151} C_VEL
LIN {X 0,Y 282.567,Z 595.653,A -85,B 0,C 180,E1 -17098.575,E2 -17098.575} C_VEL
LIN {X 0,Y 282.458,Z 594.367,A -85,B 0,C 180,E1 -17100,E2 -17100} C_VEL
LIN {X 0,Y 282.479,Z 591.568,A -85,B 0,C 180,E1 -17102.139,E2 -17102.139} C_VEL
LIN {X 0,Y 282.617,Z 587.678,A -85,B 0,C 180,E1 -17104.279,E2 -17104.279} C_VEL
LIN {X 0,Y 282.787,Z 582.585,A -85,B 0,C 180,E1 -17106.421,E2 -17106.421} C_VEL
LIN {X 0,Y 283.153,Z 576.134,A -85,B 0,C 180,E1 -17108.565,E2 -17108.565} C_VEL
LIN {X 0,Y 283.692,Z 568.092,A -85,B 0,C 180,E1 -17110.708,E2 -17110.708} C_VEL
LIN {X 0,Y 284.458,Z 558.04,A -85,B 0,C 180,E1 -17112.848,E2 -17112.848} C_VEL
LIN {X 0,Y 285.271,Z 548.853,A -85,B 0,C 180,E1 -17114.445,E2 -17114.445} C_VEL
LIN {X 0,Y 286.167,Z 537.877,A -85,B 0,C 180,E1 -17116.003,E2 -17116.003} C_VEL
LIN {X 0,Y 287.02,Z 525.454,A -85,B 0,C 180,E1 -17117.418,E2 -17117.418} C_VEL
LIN {X 0,Y 287.851,Z 511.984,A -85,B 0,C 180,E1 -17118.598,E2 -17118.598} C_VEL
LIN {X 0,Y 288.492,Z 499.179,A -85,B 0,C 180,E1 -17119.432,E2 -17119.432} C_VEL
LIN {X 0,Y 289.122,Z 484.588,A -85,B 0,C 180,E1 -17120.081,E2 -17120.081} C_VEL
LIN {X 0,Y 291.702,Z 409.167,A -85,B 0,C 180,E1 -17122.854,E2 -17122.854} C_VEL
LIN {X 0,Y 288.345,Z 382.834,A -85,B 0,C 180,E1 -17124.005,E2 -17124.005} C_VEL
LIN {X 0,Y 288.299,Z 381.883,A -85,B 0,C 180,E1 -17124.061,E2 -17124.061} C_VEL
LIN {X 0,Y 288.181,Z 377.591,A -85,B 0,C 180,E1 -17125.026,E2 -17125.026} C_VEL
LIN {X 0,Y 285.477,Z 363.816,A -85,B 0,C 180,E1 -17128.288,E2 -17128.288} C_VEL
LIN {X 0,Y 284.396,Z 358.685,A -85,B 0,C 180,E1 -17129.518,E2 -17129.518} C_VEL
LIN {X 0,Y 284.313,Z 358.694,A -85,B 0,C 180,E1 -17132.944,E2 -17132.944} C_VEL
LIN {X 0,Y 284.325,Z 358.692,A -85,B 0,C 180,E1 -17136.387,E2 -17136.387} C_VEL
LIN {X 0,Y 284.261,Z 358.703,A -85,B 0,C 180,E1 -17140.003,E2 -17140.003} C_VEL
LIN {X 0,Y 284.24,Z 358.706,A -85,B 0,C 180,E1 -17144.187,E2 -17144.187} C_VEL
LIN {X 0,Y 284.246,Z 358.704,A -85,B 0,C 180,E1 -17148.117,E2 -17148.117} C_VEL
LIN {X 0,Y 284.314,Z 358.696,A -85,B 0,C 180,E1 -17152.281,E2 -17152.281} C_VEL
LIN {X 0,Y 286.022,Z 364.989,A -85,B 0,C 180,E1 -17154.734,E2 -17154.734} C_VEL
LIN {X 0,Y 296.973,Z 386.787,A -85,B 0,C 180,E1 -17156.85,E2 -17156.85} C_VEL
LIN {X 0,Y 304.666,Z 404.762,A -85,B 0,C 180,E1 -17158.283,E2 -17158.283} C_VEL
LIN {X 0,Y 306.078,Z 408.746,A -85,B 0,C 180,E1 -17158.554,E2 -17158.554} C_VEL
LIN {X 0,Y 303.392,Z 491.337,A -85,B 0,C 180,E1 -17160.471,E2 -17160.471} C_VEL
LIN {X 0,Y 302.617,Z 505.467,A -85,B 0,C 180,E1 -17160.856,E2 -17160.856} C_VEL
LIN {X 0,Y 301.533,Z 519.694,A -85,B 0,C 180,E1 -17161.503,E2 -17161.503} C_VEL
LIN {X 0,Y 299.992,Z 532.845,A -85,B 0,C 180,E1 -17162.343,E2 -17162.343} C_VEL
LIN {X 0,Y 298.117,Z 546.387,A -85,B 0,C 180,E1 -17163.504,E2 -17163.504} C_VEL
LIN {X 0,Y 296.107,Z 558.885,A -85,B 0,C 180,E1 -17164.894,E2 -17164.894} C_VEL
LIN {X 0,Y 293.749,Z 570.915,A -85,B 0,C 180,E1 -17166.56,E2 -17166.56} C_VEL
LIN {X 0,Y 291.779,Z 579.977,A -85,B 0,C 180,E1 -17168.076,E2 -17168.076} C_VEL
LIN {X 0,Y 289.524,Z 590.033,A -85,B 0,C 180,E1 -17170.131,E2 -17170.131} C_VEL
LIN {X 0,Y 287.595,Z 598.467,A -85,B 0,C 180,E1 -17172.238,E2 -17172.238} C_VEL
LIN {X 0,Y 285.992,Z 606.351,A -85,B 0,C 180,E1 -17174.68,E2 -17174.68} C_VEL
LIN {X 0,Y 284.417,Z 612.772,A -85,B 0,C 180,E1 -17177.148,E2 -17177.148} C_VEL
LIN {X 0,Y 283.353,Z 618.458,A -85,B 0,C 180,E1 -17180,E2 -17180} C_VEL
LIN {X 0,Y 282.728,Z 622.588,A -85,B 0,C 180,E1 -17182.858,E2 -17182.858} C_VEL
LIN {X 0,Y 282.393,Z 625.292,A -85,B 0,C 180,E1 -17185.716,E2 -17185.716} C_VEL
LIN {X 0,Y 282.31,Z 626.647,A -85,B 0,C 180,E1 -17188.571,E2 -17188.571} C_VEL
LIN {X 0,Y 282.309,Z 626.679,A -85,B 0,C 180,E1 -17191.424,E2 -17191.424} C_VEL
LIN {X 0,Y 282.387,Z 625.388,A -85,B 0,C 180,E1 -17194.28,E2 -17194.28} C_VEL
LIN {X 0,Y 282.697,Z 622.741,A -85,B 0,C 180,E1 -17197.138,E2 -17197.138} C_VEL
LIN {X 0,Y 283.338,Z 618.665,A -85,B 0,C 180,E1 -17199.997,E2 -17199.997} C_VEL
LIN {X 0,Y 284.386,Z 613.037,A -85,B 0,C 180,E1 -17202.849,E2 -17202.849} C_VEL
LIN {X 0,Y 285.939,Z 606.685,A -85,B 0,C 180,E1 -17205.318,E2 -17205.318} C_VEL
LIN {X 0,Y 287.509,Z 599.033,A -85,B 0,C 180,E1 -17207.716,E2 -17207.716} C_VEL
LIN {X 0,Y 289.44,Z 590.522,A -85,B 0,C 180,E1 -17209.871,E2 -17209.871} C_VEL
LIN {X 0,Y 291.709,Z 580.564,A -85,B 0,C 180,E1 -17211.925,E2 -17211.925} C_VEL
LIN {X 0,Y 294.081,Z 569.475,A -85,B 0,C 180,E1 -17213.781,E2 -17213.781} C_VEL
LIN {X 0,Y 296.263,Z 558.439,A -85,B 0,C 180,E1 -17215.275,E2 -17215.275} C_VEL
LIN {X 0,Y 298.167,Z 546.452,A -85,B 0,C 180,E1 -17216.603,E2 -17216.603} C_VEL
LIN {X 0,Y 300.029,Z 533.182,A -85,B 0,C 180,E1 -17217.744,E2 -17217.744} C_VEL
LIN {X 0,Y 301.591,Z 519.386,A -85,B 0,C 180,E1 -17218.628,E2 -17218.628} C_VEL
LIN {X 0,Y 302.785,Z 505.015,A -85,B 0,C 180,E1 -17219.265,E2 -17219.265} C_VEL
LIN {X 0,Y 303.646,Z 484.943,A -85,B 0,C 180,E1 -17219.793,E2 -17219.793} C_VEL
LIN {X 0,Y 306.247,Z 409.89,A -85,B 0,C 180,E1 -17221.516,E2 -17221.516} C_VEL
LIN {X 0,Y 305.412,Z 406.637,A -85,B 0,C 180,E1 -17221.7,E2 -17221.7} C_VEL
LIN {X 0,Y 298.431,Z 390.081,A -85,B 0,C 180,E1 -17222.998,E2 -17222.998} C_VEL
LIN {X 0,Y 293.178,Z 379.055,A -85,B 0,C 180,E1 -17223.987,E2 -17223.987} C_VEL
LIN {X 0,Y 291.14,Z 376.194,A -85,B 0,C 180,E1 -17224.342,E2 -17224.342} C_VEL
LIN {X 0,Y 286.565,Z 372.909,A -85,B 0,C 180,E1 -17225.068,E2 -17225.068} C_VEL
LIN {X 0,Y 281.883,Z 369.764,A -85,B 0,C 180,E1 -17225.837,E2 -17225.837} C_VEL
LIN {X 0,Y 279.668,Z 367.085,A -85,B 0,C 180,E1 -17226.25,E2 -17226.25} C_VEL
LIN {X 0,Y 278.754,Z 364.994,A -85,B 0,C 180,E1 -17226.49,E2 -17226.49} C_VEL
LIN {X 0,Y 277.196,Z 359.582,A -85,B 0,C 180,E1 -17228.706,E2 -17228.706} C_VEL
LIN {X 0,Y 277.182,Z 359.582,A -85,B 0,C 180,E1 -17233.2,E2 -17233.2} C_VEL
LIN {X 0,Y 277.183,Z 359.584,A -85,B 0,C 180,E1 -17237.328,E2 -17237.328} C_VEL
LIN {X 0,Y 277.239,Z 359.56,A -85,B 0,C 180,E1 -17241.795,E2 -17241.795} C_VEL
LIN {X 0,Y 277.266,Z 359.572,A -85,B 0,C 180,E1 -17244.339,E2 -17244.339} C_VEL
LIN {X 0,Y 277.228,Z 359.558,A -85,B 0,C 180,E1 -17247.834,E2 -17247.834} C_VEL
LIN {X 0,Y 277.227,Z 359.573,A -85,B 0,C 180,E1 -17251.205,E2 -17251.205} C_VEL
LIN {X 0,Y 277.233,Z 359.554,A -85,B 0,C 180,E1 -17254.471,E2 -17254.471} C_VEL
LIN {X 0,Y 277.246,Z 359.573,A -85,B 0,C 180,E1 -17257.651,E2 -17257.651} C_VEL
LIN {X 0,Y 277.272,Z 359.542,A -85,B 0,C 180,E1 -17260.761,E2 -17260.761} C_VEL
LIN {X 0,Y 277.396,Z 359.554,A -85,B 0,C 180,E1 -17265.324,E2 -17265.324} C_VEL
LIN {X 0,Y 277.444,Z 359.549,A -85,B 0,C 180,E1 -17269.786,E2 -17269.786} C_VEL
LIN {X 0,Y 277.585,Z 359.533,A -85,B 0,C 180,E1 -17272.727,E2 -17272.727} C_VEL
LIN {X 0,Y 277.791,Z 359.504,A -85,B 0,C 180,E1 -17278.55,E2 -17278.55} C_VEL
LIN {X 0,Y 277.798,Z 359.505,A -85,B 0,C 180,E1 -17281.45,E2 -17281.45} C_VEL
LIN {X 0,Y 277.586,Z 359.53,A -85,B 0,C 180,E1 -17287.273,E2 -17287.273} C_VEL
LIN {X 0,Y 277.443,Z 359.549,A -85,B 0,C 180,E1 -17290.214,E2 -17290.214} C_VEL
LIN {X 0,Y 277.396,Z 359.558,A -85,B 0,C 180,E1 -17294.676,E2 -17294.676} C_VEL
LIN {X 0,Y 277.272,Z 359.57,A -85,B 0,C 180,E1 -17299.239,E2 -17299.239} C_VEL
LIN {X 0,Y 277.242,Z 359.562,A -85,B 0,C 180,E1 -17303.928,E2 -17303.928} C_VEL
LIN {X 0,Y 277.223,Z 359.567,A -85,B 0,C 180,E1 -17307.47,E2 -17307.47} C_VEL
LIN {X 0,Y 277.216,Z 359.568,A -85,B 0,C 180,E1 -17310.467,E2 -17310.467} C_VEL
LIN {X 0,Y 277.234,Z 359.573,A -85,B 0,C 180,E1 -17313.897,E2 -17313.897} C_VEL
LIN {X 0,Y 277.239,Z 359.577,A -85,B 0,C 180,E1 -17317.474,E2 -17317.474} C_VEL
LIN {X 0,Y 277.173,Z 359.581,A -85,B 0,C 180,E1 -17321.243,E2 -17321.243} C_VEL
LIN {X 0,Y 277.164,Z 359.586,A -85,B 0,C 180,E1 -17325.234,E2 -17325.234} C_VEL
LIN {X 0,Y 277.175,Z 359.589,A -85,B 0,C 180,E1 -17328.761,E2 -17328.761} C_VEL
LIN {X 0,Y 277.253,Z 359.607,A -85,B 0,C 180,E1 -17330.034,E2 -17330.034} C_VEL
LIN {X 0,Y 279.859,Z 369.263,A -85,B 0,C 180,E1 -17333.759,E2 -17333.759} C_VEL
LIN {X 0,Y 288.131,Z 385.638,A -85,B 0,C 180,E1 -17335.44,E2 -17335.44} C_VEL
LIN {X 0,Y 295.547,Z 402.083,A -85,B 0,C 180,E1 -17336.891,E2 -17336.891} C_VEL
LIN {X 0,Y 298.484,Z 409.773,A -85,B 0,C 180,E1 -17337.472,E2 -17337.472} C_VEL
LIN {X 0,Y 299.895,Z 418.533,A -85,B 0,C 180,E1 -17337.887,E2 -17337.887} C_VEL
LIN {X 0,Y 296.754,Z 506.584,A -85,B 0,C 180,E1 -17339.983,E2 -17339.983} C_VEL
LIN {X 0,Y 295.573,Z 520.574,A -85,B 0,C 180,E1 -17340.537,E2 -17340.537} C_VEL
LIN {X 0,Y 294.03,Z 534.224,A -85,B 0,C 180,E1 -17341.347,E2 -17341.347} C_VEL
LIN {X 0,Y 292.114,Z 547.492,A -85,B 0,C 180,E1 -17342.413,E2 -17342.413} C_VEL
LIN {X 0,Y 290.084,Z 559.755,A -85,B 0,C 180,E1 -17343.691,E2 -17343.691} C_VEL
LIN {X 0,Y 287.797,Z 571.893,A -85,B 0,C 180,E1 -17345.282,E2 -17345.282} C_VEL
LIN {X 0,Y 285.152,Z 583.518,A -85,B 0,C 180,E1 -17347.161,E2 -17347.161} C_VEL
LIN {X 0,Y 282.768,Z 593.916,A -85,B 0,C 180,E1 -17349.26,E2 -17349.26} C_VEL
LIN {X 0,Y 280.701,Z 602.494,A -85,B 0,C 180,E1 -17351.386,E2 -17351.386} C_VEL
LIN {X 0,Y 278.898,Z 610.708,A -85,B 0,C 180,E1 -17353.91,E2 -17353.91} C_VEL
LIN {X 0,Y 277.62,Z 616.459,A -85,B 0,C 180,E1 -17356.087,E2 -17356.087} C_VEL
LIN {X 0,Y 276.543,Z 621.168,A -85,B 0,C 180,E1 -17358.272,E2 -17358.272} C_VEL
LIN {X 0,Y 275.731,Z 626.055,A -85,B 0,C 180,E1 -17361.205,E2 -17361.205} C_VEL
LIN {X 0,Y 275.298,Z 629.45,A -85,B 0,C 180,E1 -17364.141,E2 -17364.141} C_VEL
LIN {X 0,Y 275.21,Z 631.454,A -85,B 0,C 180,E1 -17367.075,E2 -17367.075} C_VEL
LIN {X 0,Y 275.218,Z 632.112,A -85,B 0,C 180,E1 -17370.002,E2 -17370.002} C_VEL
LIN {X 0,Y 275.211,Z 631.436,A -85,B 0,C 180,E1 -17372.93,E2 -17372.93} C_VEL
LIN {X 0,Y 275.336,Z 629.415,A -85,B 0,C 180,E1 -17375.862,E2 -17375.862} C_VEL
LIN {X 0,Y 275.762,Z 626.007,A -85,B 0,C 180,E1 -17378.798,E2 -17378.798} C_VEL
LIN {X 0,Y 276.546,Z 621.108,A -85,B 0,C 180,E1 -17381.733,E2 -17381.733} C_VEL
LIN {X 0,Y 278.062,Z 614.568,A -85,B 0,C 180,E1 -17384.642,E2 -17384.642} C_VEL
LIN {X 0,Y 279.645,Z 607.068,A -85,B 0,C 180,E1 -17387.252,E2 -17387.252} C_VEL
LIN {X 0,Y 281.694,Z 598.274,A -85,B 0,C 180,E1 -17389.685,E2 -17389.685} C_VEL
LIN {X 0,Y 283.956,Z 588.817,A -85,B 0,C 180,E1 -17391.795,E2 -17391.795} C_VEL
LIN {X 0,Y 288.207,Z 572.393,A -85,B 0,C 180,E1 -17394.877,E2 -17394.877} C_VEL
LIN {X 0,Y 291.174,Z 561.104,A -85,B 0,C 180,E1 -17396.601,E2 -17396.601} C_VEL
LIN {X 0,Y 294.136,Z 548.368,A -85,B 0,C 180,E1 -17398.16,E2 -17398.16} C_VEL
LIN {X 0,Y 297.028,Z 535.003,A -85,B 0,C 180,E1 -17399.406,E2 -17399.406} C_VEL
LIN {X 0,Y 299.563,Z 521.116,A -85,B 0,C 180,E1 -17400.391,E2 -17400.391} C_VEL
LIN {X 0,Y 301.805,Z 505.732,A -85,B 0,C 180,E1 -17401.16,E2 -17401.16} C_VEL
LIN {X 0,Y 309.082,Z 455.607,A -85,B 0,C 180,E1 -17403.349,E2 -17403.349} C_VEL
LIN {X 0,Y 314.439,Z 421.129,A -85,B 0,C 180,E1 -17404.843,E2 -17404.843} C_VEL
LIN {X 0,Y 314.318,Z 419.265,A -85,B 0,C 180,E1 -17405.086,E2 -17405.086} C_VEL
LIN {X 0,Y 312.484,Z 412.49,A -85,B 0,C 180,E1 -17406.658,E2 -17406.658} C_VEL
LIN {X 0,Y 309.654,Z 408.334,A -85,B 0,C 180,E1 -17408.798,E2 -17408.798} C_VEL
LIN {X 0,Y 307.343,Z 405.411,A -85,B 0,C 180,E1 -17411.231,E2 -17411.231} C_VEL
LIN {X 0,Y 306.034,Z 404.256,A -85,B 0,C 180,E1 -17413.549,E2 -17413.549} C_VEL
LIN {X 0,Y 305.759,Z 404.285,A -85,B 0,C 180,E1 -17416.405,E2 -17416.405} C_VEL
LIN {X 0,Y 306.54,Z 405.826,A -85,B 0,C 180,E1 -17418.777,E2 -17418.777} C_VEL
LIN {X 0,Y 308.719,Z 409.891,A -85,B 0,C 180,E1 -17421.686,E2 -17421.686} C_VEL
LIN {X 0,Y 311.179,Z 414.836,A -85,B 0,C 180,E1 -17423.844,E2 -17423.844} C_VEL
LIN {X 0,Y 313.09,Z 419.049,A -85,B 0,C 180,E1 -17425.212,E2 -17425.212} C_VEL
LIN {X 0,Y 315.338,Z 424.396,A -85,B 0,C 180,E1 -17426.633,E2 -17426.633} C_VEL
LIN {X 0,Y 316.735,Z 428.26,A -85,B 0,C 180,E1 -17427.46,E2 -17427.46} C_VEL
LIN {X 0,Y 306.458,Z 502.017,A -85,B 0,C 180,E1 -17430.619,E2 -17430.619} C_VEL
LIN {X 0,Y 304.067,Z 516.183,A -85,B 0,C 180,E1 -17431.529,E2 -17431.529} C_VEL
LIN {X 0,Y 301.503,Z 528.468,A -85,B 0,C 180,E1 -17432.589,E2 -17432.589} C_VEL
LIN {X 0,Y 298.633,Z 540.292,A -85,B 0,C 180,E1 -17433.893,E2 -17433.893} C_VEL
LIN {X 0,Y 295.484,Z 551.262,A -85,B 0,C 180,E1 -17435.403,E2 -17435.403} C_VEL
LIN {X 0,Y 292.467,Z 560.71,A -85,B 0,C 180,E1 -17437.015,E2 -17437.015} C_VEL
LIN {X 0,Y 289.226,Z 569.966,A -85,B 0,C 180,E1 -17438.997,E2 -17438.997} C_VEL
LIN {X 0,Y 286.265,Z 577.528,A -85,B 0,C 180,E1 -17441.017,E2 -17441.017} C_VEL
LIN {X 0,Y 283.369,Z 584.518,A -85,B 0,C 180,E1 -17443.428,E2 -17443.428} C_VEL
LIN {X 0,Y 281.292,Z 589.167,A -85,B 0,C 180,E1 -17445.532,E2 -17445.532} C_VEL
LIN {X 0,Y 279.414,Z 592.732,A -85,B 0,C 180,E1 -17447.655,E2 -17447.655} C_VEL
LIN {X 0,Y 278.194,Z 595.236,A -85,B 0,C 180,E1 -17449.814,E2 -17449.814} C_VEL
LIN {X 0,Y 277.371,Z 596.387,A -85,B 0,C 180,E1 -17451.256,E2 -17451.256} C_VEL
LIN {X 0,Y 276.738,Z 597.13,A -85,B 0,C 180,E1 -17452.705,E2 -17452.705} C_VEL
LIN {X 0,Y 276.247,Z 597.411,A -85,B 0,C 180,E1 -17454.159,E2 -17454.159} C_VEL
LIN {X 0,Y 275.935,Z 597.271,A -85,B 0,C 180,E1 -17455.618,E2 -17455.618} C_VEL
LIN {X 0,Y 275.683,Z 596.728,A -85,B 0,C 180,E1 -17457.078,E2 -17457.078} C_VEL
LIN {X 0,Y 275.487,Z 595.751,A -85,B 0,C 180,E1 -17458.538,E2 -17458.538} C_VEL
LIN {X 0,Y 275.377,Z 594.313,A -85,B 0,C 180,E1 -17460,E2 -17460} C_VEL
LIN {X 0,Y 275.407,Z 591.327,A -85,B 0,C 180,E1 -17462.194,E2 -17462.194} C_VEL
LIN {X 0,Y 275.517,Z 587.243,A -85,B 0,C 180,E1 -17464.389,E2 -17464.389} C_VEL
LIN {X 0,Y 275.728,Z 581.939,A -85,B 0,C 180,E1 -17466.586,E2 -17466.586} C_VEL
LIN {X 0,Y 276.108,Z 575.245,A -85,B 0,C 180,E1 -17468.785,E2 -17468.785} C_VEL
LIN {X 0,Y 276.695,Z 566.866,A -85,B 0,C 180,E1 -17470.982,E2 -17470.982} C_VEL
LIN {X 0,Y 277.328,Z 558.355,A -85,B 0,C 180,E1 -17472.811,E2 -17472.811} C_VEL
LIN {X 0,Y 278.245,Z 547.989,A -85,B 0,C 180,E1 -17474.631,E2 -17474.631} C_VEL
LIN {X 0,Y 279.137,Z 536.788,A -85,B 0,C 180,E1 -17476.228,E2 -17476.228} C_VEL
LIN {X 0,Y 279.943,Z 525.405,A -85,B 0,C 180,E1 -17477.534,E2 -17477.534} C_VEL
LIN {X 0,Y 280.793,Z 512.381,A -85,B 0,C 180,E1 -17478.705,E2 -17478.705} C_VEL
LIN {X 0,Y 281.468,Z 498.889,A -85,B 0,C 180,E1 -17479.604,E2 -17479.604} C_VEL
LIN {X 0,Y 282.102,Z 484.244,A -85,B 0,C 180,E1 -17480.27,E2 -17480.27} C_VEL
LIN {X 0,Y 284.76,Z 410.098,A -85,B 0,C 180,E1 -17483.093,E2 -17483.093} C_VEL
LIN {X 0,Y 281.501,Z 384.229,A -85,B 0,C 180,E1 -17484.252,E2 -17484.252} C_VEL
LIN {X 0,Y 281.353,Z 382.074,A -85,B 0,C 180,E1 -17484.383,E2 -17484.383} C_VEL
LIN {X 0,Y 281.2,Z 378.732,A -85,B 0,C 180,E1 -17485.143,E2 -17485.143} C_VEL
LIN {X 0,Y 278.286,Z 364.04,A -85,B 0,C 180,E1 -17488.675,E2 -17488.675} C_VEL
LIN {X 0,Y 277.359,Z 359.563,A -85,B 0,C 180,E1 -17489.82,E2 -17489.82} C_VEL
LIN {X 0,Y 277.253,Z 359.572,A -85,B 0,C 180,E1 -17493.895,E2 -17493.895} C_VEL
LIN {X 0,Y 277.239,Z 359.577,A -85,B 0,C 180,E1 -17497.474,E2 -17497.474} C_VEL
LIN {X 0,Y 277.183,Z 359.582,A -85,B 0,C 180,E1 -17501.242,E2 -17501.242} C_VEL
LIN {X 0,Y 277.18,Z 359.584,A -85,B 0,C 180,E1 -17505.231,E2 -17505.231} C_VEL
LIN {X 0,Y 277.19,Z 359.582,A -85,B 0,C 180,E1 -17508.758,E2 -17508.758} C_VEL
LIN {X 0,Y 277.269,Z 359.725,A -85,B 0,C 180,E1 -17511.531,E2 -17511.531} C_VEL
LIN {X 0,Y 278.849,Z 365.242,A -85,B 0,C 180,E1 -17513.701,E2 -17513.701} C_VEL
LIN {X 0,Y 289.282,Z 385.529,A -85,B 0,C 180,E1 -17515.809,E2 -17515.809} C_VEL
LIN {X 0,Y 296.409,Z 401.281,A -85,B 0,C 180,E1 -17517.189,E2 -17517.189} C_VEL
LIN {X 0,Y 300.008,Z 410.307,A -85,B 0,C 180,E1 -17517.883,E2 -17517.883} C_VEL
LIN {X 0,Y 297.215,Z 491.947,A -85,B 0,C 180,E1 -17519.808,E2 -17519.808} C_VEL
LIN {X 0,Y 296.374,Z 506.689,A -85,B 0,C 180,E1 -17520.23,E2 -17520.23} C_VEL
LIN {X 0,Y 295.245,Z 520.533,A -85,B 0,C 180,E1 -17520.888,E2 -17520.888} C_VEL
LIN {X 0,Y 293.589,Z 534.043,A -85,B 0,C 180,E1 -17521.783,E2 -17521.783} C_VEL
LIN {X 0,Y 291.566,Z 547.742,A -85,B 0,C 180,E1 -17523.015,E2 -17523.015} C_VEL
LIN {X 0,Y 289.424,Z 560.247,A -85,B 0,C 180,E1 -17524.466,E2 -17524.466} C_VEL
LIN {X 0,Y 287.006,Z 572.054,A -85,B 0,C 180,E1 -17526.167,E2 -17526.167} C_VEL
LIN {X 0,Y 284.778,Z 581.827,A -85,B 0,C 180,E1 -17527.89,E2 -17527.89} C_VEL
LIN {X 0,Y 282.454,Z 591.585,A -85,B 0,C 180,E1 -17529.991,E2 -17529.991} C_VEL
LIN {X 0,Y 280.493,Z 599.926,A -85,B 0,C 180,E1 -17532.2,E2 -17532.2} C_VEL
LIN {X 0,Y 278.866,Z 607.425,A -85,B 0,C 180,E1 -17534.653,E2 -17534.653} C_VEL
LIN {X 0,Y 277.464,Z 612.841,A -85,B 0,C 180,E1 -17536.821,E2 -17536.821} C_VEL
LIN {X 0,Y 276.338,Z 618.527,A -85,B 0,C 180,E1 -17539.743,E2 -17539.743} C_VEL
LIN {X 0,Y 275.677,Z 622.656,A -85,B 0,C 180,E1 -17542.675,E2 -17542.675} C_VEL
LIN {X 0,Y 275.307,Z 625.36,A -85,B 0,C 180,E1 -17545.606,E2 -17545.606} C_VEL
LIN {X 0,Y 275.237,Z 626.714,A -85,B 0,C 180,E1 -17548.535,E2 -17548.535} C_VEL
LIN {X 0,Y 275.236,Z 626.746,A -85,B 0,C 180,E1 -17551.461,E2 -17551.461} C_VEL
LIN {X 0,Y 275.302,Z 625.455,A -85,B 0,C 180,E1 -17554.39,E2 -17554.39} C_VEL
LIN {X 0,Y 275.49,Z 624.303,A -85,B 0,C 180,E1 -17555.855,E2 -17555.855} C_VEL
LIN {X 0,Y 275.928,Z 620.955,A -85,B 0,C 180,E1 -17558.788,E2 -17558.788} C_VEL
LIN {X 0,Y 276.851,Z 616.12,A -85,B 0,C 180,E1 -17561.715,E2 -17561.715} C_VEL
LIN {X 0,Y 277.865,Z 611.459,A -85,B 0,C 180,E1 -17563.901,E2 -17563.901} C_VEL
LIN {X 0,Y 279.465,Z 604.682,A -85,B 0,C 180,E1 -17566.432,E2 -17566.432} C_VEL
LIN {X 0,Y 281.049,Z 597.738,A -85,B 0,C 180,E1 -17568.552,E2 -17568.552} C_VEL
LIN {X 0,Y 283.136,Z 589.09,A -85,B 0,C 180,E1 -17570.712,E2 -17570.712} C_VEL
LIN {X 0,Y 285.567,Z 578.763,A -85,B 0,C 180,E1 -17572.804,E2 -17572.804} C_VEL
LIN {X 0,Y 288.078,Z 567.211,A -85,B 0,C 180,E1 -17574.692,E2 -17574.692} C_VEL
LIN {X 0,Y 290.466,Z 554.697,A -85,B 0,C 180,E1 -17576.334,E2 -17576.334} C_VEL
LIN {X 0,Y 292.318,Z 542.993,A -85,B 0,C 180,E1 -17577.566,E2 -17577.566} C_VEL
LIN {X 0,Y 294.19,Z 529.854,A -85,B 0,C 180,E1 -17578.636,E2 -17578.636} C_VEL
LIN {X 0,Y 295.76,Z 515.636,A -85,B 0,C 180,E1 -17579.491,E2 -17579.491} C_VEL
LIN {X 0,Y 296.831,Z 501.611,A -85,B 0,C 180,E1 -17580.058,E2 -17580.058} C_VEL
LIN {X 0,Y 298.859,Z 446.967,A -85,B 0,C 180,E1 -17581.362,E2 -17581.362} C_VEL
LIN {X 0,Y 300.056,Z 410.416,A -85,B 0,C 180,E1 -17582.231,E2 -17582.231} C_VEL
LIN {X 0,Y 293.455,Z 394.444,A -85,B 0,C 180,E1 -17583.506,E2 -17583.506} C_VEL
LIN {X 0,Y 286.452,Z 379.786,A -85,B 0,C 180,E1 -17584.878,E2 -17584.878} C_VEL
LIN {X 0,Y 280.262,Z 368.169,A -85,B 0,C 180,E1 -17586.127,E2 -17586.127} C_VEL
LIN {X 0,Y 279.668,Z 367.085,A -85,B 0,C 180,E1 -17586.25,E2 -17586.25} C_VEL
LIN {X 0,Y 277.952,Z 365.301,A -85,B 0,C 180,E1 -17586.628,E2 -17586.628} C_VEL
LIN {X 0,Y 273.711,Z 363.669,A -85,B 0,C 180,E1 -17587.773,E2 -17587.773} C_VEL
LIN {X 0,Y 271.179,Z 362.018,A -85,B 0,C 180,E1 -17588.809,E2 -17588.809} C_VEL
LIN {X 0,Y 270.165,Z 360.549,A -85,B 0,C 180,E1 -17589.735,E2 -17589.735} C_VEL
LIN {X 0,Y 270.118,Z 360.461,A -85,B 0,C 180,E1 -17589.964,E2 -17589.964} C_VEL
LIN {X 0,Y 270.139,Z 360.46,A -85,B 0,C 180,E1 -17593.243,E2 -17593.243} C_VEL
LIN {X 0,Y 270.142,Z 360.461,A -85,B 0,C 180,E1 -17597.436,E2 -17597.436} C_VEL
LIN {X 0,Y 270.182,Z 360.441,A -85,B 0,C 180,E1 -17601.37,E2 -17601.37} C_VEL
LIN {X 0,Y 270.187,Z 360.452,A -85,B 0,C 180,E1 -17605.092,E2 -17605.092} C_VEL
LIN {X 0,Y 270.173,Z 360.449,A -85,B 0,C 180,E1 -17609.135,E2 -17609.135} C_VEL
LIN {X 0,Y 270.211,Z 360.435,A -85,B 0,C 180,E1 -17612.162,E2 -17612.162} C_VEL
LIN {X 0,Y 270.215,Z 360.442,A -85,B 0,C 180,E1 -17615.541,E2 -17615.541} C_VEL
LIN {X 0,Y 270.211,Z 360.422,A -85,B 0,C 180,E1 -17620.237,E2 -17620.237} C_VEL
LIN {X 0,Y 270.355,Z 360.434,A -85,B 0,C 180,E1 -17624.932,E2 -17624.932} C_VEL
LIN {X 0,Y 270.396,Z 360.427,A -85,B 0,C 180,E1 -17629.517,E2 -17629.517} C_VEL
LIN {X 0,Y 270.547,Z 360.408,A -85,B 0,C 180,E1 -17632.537,E2 -17632.537} C_VEL
LIN {X 0,Y 270.756,Z 360.381,A -85,B 0,C 180,E1 -17638.512,E2 -17638.512} C_VEL
LIN {X 0,Y 270.762,Z 360.381,A -85,B 0,C 180,E1 -17641.487,E2 -17641.487} C_VEL
LIN {X 0,Y 270.548,Z 360.406,A -85,B 0,C 180,E1 -17647.463,E2 -17647.463} C_VEL
LIN {X 0,Y 270.396,Z 360.429,A -85,B 0,C 180,E1 -17650.483,E2 -17650.483} C_VEL
LIN {X 0,Y 270.355,Z 360.432,A -85,B 0,C 180,E1 -17655.067,E2 -17655.067} C_VEL
LIN {X 0,Y 270.21,Z 360.448,A -85,B 0,C 180,E1 -17659.762,E2 -17659.762} C_VEL
LIN {X 0,Y 270.169,Z 360.447,A -85,B 0,C 180,E1 -17664.437,E2 -17664.437} C_VEL
LIN {X 0,Y 270.172,Z 360.439,A -85,B 0,C 180,E1 -17667.92,E2 -17667.92} C_VEL
LIN {X 0,Y 270.157,Z 360.457,A -85,B 0,C 180,E1 -17671.352,E2 -17671.352} C_VEL
LIN {X 0,Y 270.186,Z 360.454,A -85,B 0,C 180,E1 -17674.908,E2 -17674.908} C_VEL
LIN {X 0,Y 270.187,Z 360.452,A -85,B 0,C 180,E1 -17678.712,E2 -17678.712} C_VEL
LIN {X 0,Y 270.137,Z 360.459,A -85,B 0,C 180,E1 -17683.247,E2 -17683.247} C_VEL
LIN {X 0,Y 270.141,Z 360.463,A -85,B 0,C 180,E1 -17687.439,E2 -17687.439} C_VEL
LIN {X 0,Y 270.164,Z 360.52,A -85,B 0,C 180,E1 -17689.129,E2 -17689.129} C_VEL
LIN {X 0,Y 272.669,Z 369.313,A -85,B 0,C 180,E1 -17692.647,E2 -17692.647} C_VEL
LIN {X 0,Y 281.731,Z 386.845,A -85,B 0,C 180,E1 -17694.577,E2 -17694.577} C_VEL
LIN {X 0,Y 289.487,Z 403.918,A -85,B 0,C 180,E1 -17696.161,E2 -17696.161} C_VEL
LIN {X 0,Y 292.736,Z 412.394,A -85,B 0,C 180,E1 -17696.829,E2 -17696.829} C_VEL
LIN {X 0,Y 293.849,Z 419.902,A -85,B 0,C 180,E1 -17697.184,E2 -17697.184} C_VEL
LIN {X 0,Y 290.639,Z 506.583,A -85,B 0,C 180,E1 -17699.286,E2 -17699.286} C_VEL
LIN {X 0,Y 289.339,Z 521.278,A -85,B 0,C 180,E1 -17699.888,E2 -17699.888} C_VEL
LIN {X 0,Y 287.664,Z 535.293,A -85,B 0,C 180,E1 -17700.752,E2 -17700.752} C_VEL
LIN {X 0,Y 285.535,Z 549.198,A -85,B 0,C 180,E1 -17701.921,E2 -17701.921} C_VEL
LIN {X 0,Y 283.321,Z 561.878,A -85,B 0,C 180,E1 -17703.318,E2 -17703.318} C_VEL
LIN {X 0,Y 280.825,Z 574.174,A -85,B 0,C 180,E1 -17705.022,E2 -17705.022} C_VEL
LIN {X 0,Y 278.173,Z 585.343,A -85,B 0,C 180,E1 -17706.948,E2 -17706.948} C_VEL
LIN {X 0,Y 275.74,Z 595.366,A -85,B 0,C 180,E1 -17709.097,E2 -17709.097} C_VEL
LIN {X 0,Y 273.654,Z 603.69,A -85,B 0,C 180,E1 -17711.278,E2 -17711.278} C_VEL
LIN {X 0,Y 271.777,Z 611.65,A -85,B 0,C 180,E1 -17713.862,E2 -17713.862} C_VEL
LIN {X 0,Y 270.267,Z 618.056,A -85,B 0,C 180,E1 -17716.468,E2 -17716.468} C_VEL
LIN {X 0,Y 269.075,Z 623.74,A -85,B 0,C 180,E1 -17719.468,E2 -17719.468} C_VEL
LIN {X 0,Y 268.407,Z 627.865,A -85,B 0,C 180,E1 -17722.48,E2 -17722.48} C_VEL
LIN {X 0,Y 268.13,Z 630.555,A -85,B 0,C 180,E1 -17725.492,E2 -17725.492} C_VEL
LIN {X 0,Y 268.126,Z 631.882,A -85,B 0,C 180,E1 -17728.5,E2 -17728.5} C_VEL
LIN {X 0,Y 268.126,Z 631.874,A -85,B 0,C 180,E1 -17731.504,E2 -17731.504} C_VEL
LIN {X 0,Y 268.142,Z 630.527,A -85,B 0,C 180,E1 -17734.512,E2 -17734.512} C_VEL
LIN {X 0,Y 268.426,Z 627.821,A -85,B 0,C 180,E1 -17737.524,E2 -17737.524} C_VEL
LIN {X 0,Y 269.079,Z 623.684,A -85,B 0,C 180,E1 -17740.537,E2 -17740.537} C_VEL
LIN {X 0,Y 270.271,Z 617.986,A -85,B 0,C 180,E1 -17743.537,E2 -17743.537} C_VEL
LIN {X 0,Y 271.776,Z 611.559,A -85,B 0,C 180,E1 -17746.142,E2 -17746.142} C_VEL
LIN {X 0,Y 273.612,Z 603.577,A -85,B 0,C 180,E1 -17748.73,E2 -17748.73} C_VEL
LIN {X 0,Y 275.743,Z 595.25,A -85,B 0,C 180,E1 -17750.907,E2 -17750.907} C_VEL
LIN {X 0,Y 279.853,Z 581.952,A -85,B 0,C 180,E1 -17754.087,E2 -17754.087} C_VEL
LIN {X 0,Y 283.257,Z 571.054,A -85,B 0,C 180,E1 -17756.132,E2 -17756.132} C_VEL
LIN {X 0,Y 286.393,Z 560.199,A -85,B 0,C 180,E1 -17757.793,E2 -17757.793} C_VEL
LIN {X 0,Y 289.456,Z 548.384,A -85,B 0,C 180,E1 -17759.253,E2 -17759.253} C_VEL
LIN {X 0,Y 292.589,Z 535.361,A -85,B 0,C 180,E1 -17760.494,E2 -17760.494} C_VEL
LIN {X 0,Y 295.519,Z 520.73,A -85,B 0,C 180,E1 -17761.549,E2 -17761.549} C_VEL
LIN {X 0,Y 297.97,Z 505.669,A -85,B 0,C 180,E1 -17762.304,E2 -17762.304} C_VEL
LIN {X 0,Y 305.616,Z 456.475,A -85,B 0,C 180,E1 -17764.493,E2 -17764.493} C_VEL
LIN {X 0,Y 311.112,Z 423.835,A -85,B 0,C 180,E1 -17765.897,E2 -17765.897} C_VEL
LIN {X 0,Y 309.862,Z 418.565,A -85,B 0,C 180,E1 -17767.144,E2 -17767.144} C_VEL
LIN {X 0,Y 307.255,Z 414.584,A -85,B 0,C 180,E1 -17769.308,E2 -17769.308} C_VEL
LIN {X 0,Y 305.303,Z 412.041,A -85,B 0,C 180,E1 -17771.61,E2 -17771.61} C_VEL
LIN {X 0,Y 304.18,Z 411.077,A -85,B 0,C 180,E1 -17773.882,E2 -17773.882} C_VEL
LIN {X 0,Y 304.021,Z 411.197,A -85,B 0,C 180,E1 -17776.517,E2 -17776.517} C_VEL
LIN {X 0,Y 304.674,Z 412.651,A -85,B 0,C 180,E1 -17778.633,E2 -17778.633} C_VEL
LIN {X 0,Y 306.516,Z 416.414,A -85,B 0,C 180,E1 -17781.346,E2 -17781.346} C_VEL
LIN {X 0,Y 308.823,Z 421.419,A -85,B 0,C 180,E1 -17783.544,E2 -17783.544} C_VEL
LIN {X 0,Y 310.895,Z 426.338,A -85,B 0,C 180,E1 -17785.118,E2 -17785.118} C_VEL
LIN {X 0,Y 312.827,Z 431.689,A -85,B 0,C 180,E1 -17786.447,E2 -17786.447} C_VEL
LIN {X 0,Y 302.205,Z 502.886,A -85,B 0,C 180,E1 -17789.566,E2 -17789.566} C_VEL
LIN {X 0,Y 299.614,Z 516.999,A -85,B 0,C 180,E1 -17790.489,E2 -17790.489} C_VEL
LIN {X 0,Y 296.893,Z 529.059,A -85,B 0,C 180,E1 -17791.55,E2 -17791.55} C_VEL
LIN {X 0,Y 294.094,Z 539.784,A -85,B 0,C 180,E1 -17792.736,E2 -17792.736} C_VEL
LIN {X 0,Y 290.801,Z 550.633,A -85,B 0,C 180,E1 -17794.214,E2 -17794.214} C_VEL
LIN {X 0,Y 286.922,Z 561.915,A -85,B 0,C 180,E1 -17796.162,E2 -17796.162} C_VEL
LIN {X 0,Y 283.463,Z 570.958,A -85,B 0,C 180,E1 -17798.167,E2 -17798.167} C_VEL
LIN {X 0,Y 280.262,Z 578.41,A -85,B 0,C 180,E1 -17800.213,E2 -17800.213} C_VEL
LIN {X 0,Y 277.613,Z 584.391,A -85,B 0,C 180,E1 -17802.315,E2 -17802.315} C_VEL
LIN {X 0,Y 275.242,Z 589.151,A -85,B 0,C 180,E1 -17804.448,E2 -17804.448} C_VEL
LIN {X 0,Y 273.148,Z 592.82,A -85,B 0,C 180,E1 -17806.611,E2 -17806.611} C_VEL
LIN {X 0,Y 272.098,Z 594.66,A -85,B 0,C 180,E1 -17808.075,E2 -17808.075} C_VEL
LIN {X 0,Y 271.264,Z 596.08,A -85,B 0,C 180,E1 -17809.551,E2 -17809.551} C_VEL
LIN {X 0,Y 270.399,Z 597.104,A -85,B 0,C 180,E1 -17811.028,E2 -17811.028} C_VEL
LIN {X 0,Y 269.721,Z 597.67,A -85,B 0,C 180,E1 -17812.514,E2 -17812.514} C_VEL
LIN {X 0,Y 269.199,Z 597.831,A -85,B 0,C 180,E1 -17814.006,E2 -17814.006} C_VEL
LIN {X 0,Y 268.88,Z 597.587,A -85,B 0,C 180,E1 -17815.503,E2 -17815.503} C_VEL
LIN {X 0,Y 268.613,Z 596.896,A -85,B 0,C 180,E1 -17817.001,E2 -17817.001} C_VEL
LIN {X 0,Y 268.409,Z 595.774,A -85,B 0,C 180,E1 -17818.5,E2 -17818.5} C_VEL
LIN {X 0,Y 268.275,Z 593.279,A -85,B 0,C 180,E1 -17820.751,E2 -17820.751} C_VEL
LIN {X 0,Y 268.407,Z 589.742,A -85,B 0,C 180,E1 -17823.002,E2 -17823.002} C_VEL
LIN {X 0,Y 268.454,Z 584.925,A -85,B 0,C 180,E1 -17825.305,E2 -17825.305} C_VEL
LIN {X 0,Y 268.819,Z 579.06,A -85,B 0,C 180,E1 -17827.511,E2 -17827.511} C_VEL
LIN {X 0,Y 269.269,Z 571.536,A -85,B 0,C 180,E1 -17829.768,E2 -17829.768} C_VEL
LIN {X 0,Y 269.979,Z 562.207,A -85,B 0,C 180,E1 -17832.02,E2 -17832.02} C_VEL
LIN {X 0,Y 270.878,Z 551.533,A -85,B 0,C 180,E1 -17834.078,E2 -17834.078} C_VEL
LIN {X 0,Y 271.767,Z 540.844,A -85,B 0,C 180,E1 -17835.756,E2 -17835.756} C_VEL
LIN {X 0,Y 272.673,Z 528.327,A -85,B 0,C 180,E1 -17837.322,E2 -17837.322} C_VEL
LIN {X 0,Y 273.46,Z 515.907,A -85,B 0,C 180,E1 -17838.545,E2 -17838.545} C_VEL
LIN {X 0,Y 274.244,Z 502.247,A -85,B 0,C 180,E1 -17839.558,E2 -17839.558} C_VEL
LIN {X 0,Y 274.914,Z 487.98,A -85,B 0,C 180,E1 -17840.287,E2 -17840.287} C_VEL
LIN {X 0,Y 277.763,Z 410.625,A -85,B 0,C 180,E1 -17843.351,E2 -17843.351} C_VEL
LIN {X 0,Y 274.553,Z 384.725,A -85,B 0,C 180,E1 -17844.543,E2 -17844.543} C_VEL
LIN {X 0,Y 274.406,Z 382.306,A -85,B 0,C 180,E1 -17844.695,E2 -17844.695} C_VEL
LIN {X 0,Y 273.207,Z 374.643,A -85,B 0,C 180,E1 -17846.528,E2 -17846.528} C_VEL
LIN {X 0,Y 270.306,Z 360.441,A -85,B 0,C 180,E1 -17850.057,E2 -17850.057} C_VEL
LIN {X 0,Y 270.205,Z 360.453,A -85,B 0,C 180,E1 -17854.905,E2 -17854.905} C_VEL
LIN {X 0,Y 270.174,Z 360.454,A -85,B 0,C 180,E1 -17858.701,E2 -17858.701} C_VEL
LIN {X 0,Y 270.155,Z 360.458,A -85,B 0,C 180,E1 -17863.244,E2 -17863.244} C_VEL
LIN {X 0,Y 270.158,Z 360.46,A -85,B 0,C 180,E1 -17867.437,E2 -17867.437} C_VEL
LIN {X 0,Y 270.181,Z 360.508,A -85,B 0,C 180,E1 -17870.589,E2 -17870.589} C_VEL
LIN {X 0,Y 271.592,Z 365.41,A -85,B 0,C 180,E1 -17872.57,E2 -17872.57} C_VEL
LIN {X 0,Y 273.752,Z 369.295,A -85,B 0,C 180,E1 -17873.042,E2 -17873.042} C_VEL
LIN {X 0,Y 281.028,Z 383.167,A -85,B 0,C 180,E1 -17874.581,E2 -17874.581} C_VEL
LIN {X 0,Y 288.265,Z 398.315,A -85,B 0,C 180,E1 -17876.048,E2 -17876.048} C_VEL
LIN {X 0,Y 293.96,Z 412.199,A -85,B 0,C 180,E1 -17877.192,E2 -17877.192} C_VEL
LIN {X 0,Y 291.092,Z 492.558,A -85,B 0,C 180,E1 -17879.119,E2 -17879.119} C_VEL
LIN {X 0,Y 290.245,Z 506.772,A -85,B 0,C 180,E1 -17879.535,E2 -17879.535} C_VEL
LIN {X 0,Y 289.082,Z 520.611,A -85,B 0,C 180,E1 -17880.205,E2 -17880.205} C_VEL
LIN {X 0,Y 287.356,Z 534.118,A -85,B 0,C 180,E1 -17881.114,E2 -17881.114} C_VEL
LIN {X 0,Y 285.408,Z 546.806,A -85,B 0,C 180,E1 -17882.258,E2 -17882.258} C_VEL
LIN {X 0,Y 283.307,Z 559.028,A -85,B 0,C 180,E1 -17883.675,E2 -17883.675} C_VEL
LIN {X 0,Y 280.774,Z 571.057,A -85,B 0,C 180,E1 -17885.407,E2 -17885.407} C_VEL
LIN {X 0,Y 278.618,Z 580.118,A -85,B 0,C 180,E1 -17886.982,E2 -17886.982} C_VEL
LIN {X 0,Y 276.175,Z 590.173,A -85,B 0,C 180,E1 -17889.127,E2 -17889.127} C_VEL
LIN {X 0,Y 274.054,Z 598.522,A -85,B 0,C 180,E1 -17891.302,E2 -17891.302} C_VEL
LIN {X 0,Y 272.271,Z 606.489,A -85,B 0,C 180,E1 -17893.888,E2 -17893.888} C_VEL
LIN {X 0,Y 270.525,Z 612.91,A -85,B 0,C 180,E1 -17896.476,E2 -17896.476} C_VEL
LIN {X 0,Y 269.325,Z 618.595,A -85,B 0,C 180,E1 -17899.473,E2 -17899.473} C_VEL
LIN {X 0,Y 268.622,Z 622.724,A -85,B 0,C 180,E1 -17902.481,E2 -17902.481} C_VEL
LIN {X 0,Y 268.224,Z 625.427,A -85,B 0,C 180,E1 -17905.489,E2 -17905.489} C_VEL
LIN {X 0,Y 268.143,Z 626.782,A -85,B 0,C 180,E1 -17908.496,E2 -17908.496} C_VEL
LIN {X 0,Y 268.143,Z 626.813,A -85,B 0,C 180,E1 -17911.5,E2 -17911.5} C_VEL
LIN {X 0,Y 268.223,Z 625.522,A -85,B 0,C 180,E1 -17914.506,E2 -17914.506} C_VEL
LIN {X 0,Y 268.559,Z 622.874,A -85,B 0,C 180,E1 -17917.516,E2 -17917.516} C_VEL
LIN {X 0,Y 269.298,Z 618.798,A -85,B 0,C 180,E1 -17920.524,E2 -17920.524} C_VEL
LIN {X 0,Y 270.495,Z 613.17,A -85,B 0,C 180,E1 -17923.521,E2 -17923.521} C_VEL
LIN {X 0,Y 272.196,Z 606.817,A -85,B 0,C 180,E1 -17926.112,E2 -17926.112} C_VEL
LIN {X 0,Y 273.994,Z 598.918,A -85,B 0,C 180,E1 -17928.698,E2 -17928.698} C_VEL
LIN {X 0,Y 276.075,Z 590.652,A -85,B 0,C 180,E1 -17930.876,E2 -17930.876} C_VEL
LIN {X 0,Y 278.579,Z 580.693,A -85,B 0,C 180,E1 -17933.016,E2 -17933.016} C_VEL
LIN {X 0,Y 281.133,Z 569.602,A -85,B 0,C 180,E1 -17934.949,E2 -17934.949} C_VEL
LIN {X 0,Y 283.461,Z 558.564,A -85,B 0,C 180,E1 -17936.503,E2 -17936.503} C_VEL
LIN {X 0,Y 285.532,Z 546.576,A -85,B 0,C 180,E1 -17937.88,E2 -17937.88} C_VEL
LIN {X 0,Y 287.548,Z 533.301,A -85,B 0,C 180,E1 -17939.06,E2 -17939.06} C_VEL
LIN {X 0,Y 289.211,Z 519.5,A -85,B 0,C 180,E1 -17939.976,E2 -17939.976} C_VEL
LIN {X 0,Y 290.503,Z 505.153,A -85,B 0,C 180,E1 -17940.63,E2 -17940.63} C_VEL
LIN {X 0,Y 291.411,Z 485.435,A -85,B 0,C 180,E1 -17941.168,E2 -17941.168} C_VEL
LIN {X 0,Y 293.433,Z 430.214,A -85,B 0,C 180,E1 -17942.486,E2 -17942.486} C_VEL
LIN {X 0,Y 294.062,Z 412.392,A -85,B 0,C 180,E1 -17942.915,E2 -17942.915} C_VEL
LIN {X 0,Y 287.702,Z 397.11,A -85,B 0,C 180,E1 -17944.191,E2 -17944.191} C_VEL
LIN {X 0,Y 281,Z 383.059,A -85,B 0,C 180,E1 -17945.557,E2 -17945.557} C_VEL
LIN {X 0,Y 273.56,Z 368.984,A -85,B 0,C 180,E1 -17947.134,E2 -17947.134} C_VEL
LIN {X 0,Y 271.491,Z 365.077,A -85,B 0,C 180,E1 -17947.631,E2 -17947.631} C_VEL
LIN {X 0,Y 270.13,Z 360.461,A -85,B 0,C 180,E1 -17949.595,E2 -17949.595} C_VEL
LIN {X 0,Y 270.118,Z 360.461,A -85,B 0,C 180,E1 -17949.964,E2 -17949.964} C_VEL
LIN {X 0,Y 269.447,Z 360.546,A -85,B 0,C 180,E1 -17951.208,E2 -17951.208} C_VEL
LIN {X 0,Y 266.613,Z 360.899,A -85,B 0,C 180,E1 -17953.236,E2 -17953.236} C_VEL
LIN {X 0,Y 264.197,Z 361.2,A -85,B 0,C 180,E1 -17954.885,E2 -17954.885} C_VEL
LIN {X 0,Y 263.141,Z 361.33,A -85,B 0,C 180,E1 -17956.162,E2 -17956.162} C_VEL
LIN {X 0,Y 263.044,Z 361.339,A -85,B 0,C 180,E1 -17956.595,E2 -17956.595} C_VEL
LIN {X 0,Y 263.103,Z 361.328,A -85,B 0,C 180,E1 -17960.769,E2 -17960.769} C_VEL
LIN {X 0,Y 263.146,Z 361.33,A -85,B 0,C 180,E1 -17964.015,E2 -17964.015} C_VEL
LIN {X 0,Y 263.117,Z 361.314,A -85,B 0,C 180,E1 -17967.709,E2 -17967.709} C_VEL
LIN {X 0,Y 263.136,Z 361.321,A -85,B 0,C 180,E1 -17971.804,E2 -17971.804} C_VEL
LIN {X 0,Y 263.177,Z 361.313,A -85,B 0,C 180,E1 -17975.217,E2 -17975.217} C_VEL
LIN {X 0,Y 263.196,Z 361.3,A -85,B 0,C 180,E1 -17979.688,E2 -17979.688} C_VEL
LIN {X 0,Y 263.297,Z 361.313,A -85,B 0,C 180,E1 -17984.519,E2 -17984.519} C_VEL
LIN {X 0,Y 263.336,Z 361.307,A -85,B 0,C 180,E1 -17989.233,E2 -17989.233} C_VEL
LIN {X 0,Y 263.511,Z 361.283,A -85,B 0,C 180,E1 -17992.336,E2 -17992.336} C_VEL
LIN {X 0,Y 263.72,Z 361.257,A -85,B 0,C 180,E1 -17998.473,E2 -17998.473} C_VEL
LIN {X 0,Y 263.725,Z 361.258,A -85,B 0,C 180,E1 -18001.527,E2 -18001.527} C_VEL
LIN {X 0,Y 263.512,Z 361.283,A -85,B 0,C 180,E1 -18007.663,E2 -18007.663} C_VEL
LIN {X 0,Y 263.335,Z 361.309,A -85,B 0,C 180,E1 -18010.767,E2 -18010.767} C_VEL
LIN {X 0,Y 263.297,Z 361.311,A -85,B 0,C 180,E1 -18015.481,E2 -18015.481} C_VEL
LIN {X 0,Y 263.196,Z 361.314,A -85,B 0,C 180,E1 -18020.312,E2 -18020.312} C_VEL
LIN {X 0,Y 263.107,Z 361.335,A -85,B 0,C 180,E1 -18025.302,E2 -18025.302} C_VEL
LIN {X 0,Y 263.105,Z 361.314,A -85,B 0,C 180,E1 -18028.738,E2 -18028.738} C_VEL
LIN {X 0,Y 263.114,Z 361.335,A -85,B 0,C 180,E1 -18032.291,E2 -18032.291} C_VEL
LIN {X 0,Y 263.163,Z 361.329,A -85,B 0,C 180,E1 -18036.762,E2 -18036.762} C_VEL
LIN {X 0,Y 263.08,Z 361.341,A -85,B 0,C 180,E1 -18039.877,E2 -18039.877} C_VEL
LIN {X 0,Y 263.066,Z 361.341,A -85,B 0,C 180,E1 -18043.996,E2 -18043.996} C_VEL
LIN {X 0,Y 263.105,Z 361.487,A -85,B 0,C 180,E1 -18048.19,E2 -18048.19} C_VEL
LIN {X 0,Y 265.255,Z 369.063,A -85,B 0,C 180,E1 -18051.407,E2 -18051.407} C_VEL
LIN {X 0,Y 267.683,Z 373.427,A -85,B 0,C 180,E1 -18051.966,E2 -18051.966} C_VEL
LIN {X 0,Y 276.352,Z 390.108,A -85,B 0,C 180,E1 -18053.884,E2 -18053.884} C_VEL
LIN {X 0,Y 284.167,Z 407.533,A -85,B 0,C 180,E1 -18055.548,E2 -18055.548} C_VEL
LIN {X 0,Y 287.066,Z 415.207,A -85,B 0,C 180,E1 -18056.17,E2 -18056.17} C_VEL
LIN {X 0,Y 287.872,Z 420.058,A -85,B 0,C 180,E1 -18056.42,E2 -18056.42} C_VEL
LIN {X 0,Y 285.058,Z 494.454,A -85,B 0,C 180,E1 -18058.229,E2 -18058.229} C_VEL
LIN {X 0,Y 284.226,Z 511.061,A -85,B 0,C 180,E1 -18058.72,E2 -18058.72} C_VEL
LIN {X 0,Y 282.812,Z 525.029,A -85,B 0,C 180,E1 -18059.377,E2 -18059.377} C_VEL
LIN {X 0,Y 281.02,Z 538.623,A -85,B 0,C 180,E1 -18060.301,E2 -18060.301} C_VEL
LIN {X 0,Y 278.988,Z 550.904,A -85,B 0,C 180,E1 -18061.407,E2 -18061.407} C_VEL
LIN {X 0,Y 276.755,Z 562.996,A -85,B 0,C 180,E1 -18062.803,E2 -18062.803} C_VEL
LIN {X 0,Y 274.118,Z 575.198,A -85,B 0,C 180,E1 -18064.57,E2 -18064.57} C_VEL
LIN {X 0,Y 271.618,Z 585.278,A -85,B 0,C 180,E1 -18066.359,E2 -18066.359} C_VEL
LIN {X 0,Y 269.078,Z 595.3,A -85,B 0,C 180,E1 -18068.554,E2 -18068.554} C_VEL
LIN {X 0,Y 266.884,Z 603.624,A -85,B 0,C 180,E1 -18070.784,E2 -18070.784} C_VEL
LIN {X 0,Y 264.939,Z 611.584,A -85,B 0,C 180,E1 -18073.434,E2 -18073.434} C_VEL
LIN {X 0,Y 263.351,Z 617.99,A -85,B 0,C 180,E1 -18076.105,E2 -18076.105} C_VEL
LIN {X 0,Y 262.049,Z 623.673,A -85,B 0,C 180,E1 -18079.182,E2 -18079.182} C_VEL
LIN {X 0,Y 261.341,Z 627.798,A -85,B 0,C 180,E1 -18082.275,E2 -18082.275} C_VEL
LIN {X 0,Y 261.045,Z 630.488,A -85,B 0,C 180,E1 -18085.37,E2 -18085.37} C_VEL
LIN {X 0,Y 261.034,Z 631.815,A -85,B 0,C 180,E1 -18088.46,E2 -18088.46} C_VEL
LIN {X 0,Y 261.072,Z 631.978,A -85,B 0,C 180,E1 -18090.002,E2 -18090.002} C_VEL
LIN {X 0,Y 261.008,Z 631.3,A -85,B 0,C 180,E1 -18093.089,E2 -18093.089} C_VEL
LIN {X 0,Y 261.164,Z 629.279,A -85,B 0,C 180,E1 -18096.182,E2 -18096.182} C_VEL
LIN {X 0,Y 261.685,Z 625.87,A -85,B 0,C 180,E1 -18099.275,E2 -18099.275} C_VEL
LIN {X 0,Y 262.563,Z 620.971,A -85,B 0,C 180,E1 -18102.367,E2 -18102.367} C_VEL
LIN {X 0,Y 264.249,Z 614.43,A -85,B 0,C 180,E1 -18105.426,E2 -18105.426} C_VEL
LIN {X 0,Y 265.772,Z 607.922,A -85,B 0,C 180,E1 -18107.829,E2 -18107.829} C_VEL
LIN {X 0,Y 268.743,Z 597.298,A -85,B 0,C 180,E1 -18111.077,E2 -18111.077} C_VEL
LIN {X 0,Y 272.047,Z 588.446,A -85,B 0,C 180,E1 -18113.607,E2 -18113.607} C_VEL
LIN {X 0,Y 275.413,Z 579.14,A -85,B 0,C 180,E1 -18115.712,E2 -18115.712} C_VEL
LIN {X 0,Y 279.179,Z 567.985,A -85,B 0,C 180,E1 -18117.749,E2 -18117.749} C_VEL
LIN {X 0,Y 283.048,Z 555.388,A -85,B 0,C 180,E1 -18119.572,E2 -18119.572} C_VEL
LIN {X 0,Y 286.204,Z 544.23,A -85,B 0,C 180,E1 -18120.839,E2 -18120.839} C_VEL
LIN {X 0,Y 289.637,Z 530.493,A -85,B 0,C 180,E1 -18122.061,E2 -18122.061} C_VEL
LIN {X 0,Y 292.635,Z 515.847,A -85,B 0,C 180,E1 -18123.018,E2 -18123.018} C_VEL
LIN {X 0,Y 302.358,Z 457.991,A -85,B 0,C 180,E1 -18125.644,E2 -18125.644} C_VEL
LIN {X 0,Y 307.83,Z 427.352,A -85,B 0,C 180,E1 -18126.988,E2 -18126.988} C_VEL
LIN {X 0,Y 307.147,Z 424.38,A -85,B 0,C 180,E1 -18127.775,E2 -18127.775} C_VEL
LIN {X 0,Y 304.88,Z 420.778,A -85,B 0,C 180,E1 -18129.881,E2 -18129.881} C_VEL
LIN {X 0,Y 303.368,Z 418.765,A -85,B 0,C 180,E1 -18131.852,E2 -18131.852} C_VEL
LIN {X 0,Y 302.334,Z 417.869,A -85,B 0,C 180,E1 -18134.219,E2 -18134.219} C_VEL
LIN {X 0,Y 302.299,Z 418.224,A -85,B 0,C 180,E1 -18136.862,E2 -18136.862} C_VEL
LIN {X 0,Y 302.897,Z 419.752,A -85,B 0,C 180,E1 -18138.708,E2 -18138.708} C_VEL
LIN {X 0,Y 304.458,Z 423.141,A -85,B 0,C 180,E1 -18141.107,E2 -18141.107} C_VEL
LIN {X 0,Y 306.303,Z 427.516,A -85,B 0,C 180,E1 -18143.053,E2 -18143.053} C_VEL
LIN {X 0,Y 308.162,Z 432.383,A -85,B 0,C 180,E1 -18144.649,E2 -18144.649} C_VEL
LIN {X 0,Y 309.131,Z 435.597,A -85,B 0,C 180,E1 -18145.434,E2 -18145.434} C_VEL
LIN {X 0,Y 298.333,Z 502.926,A -85,B 0,C 180,E1 -18148.413,E2 -18148.413} C_VEL
LIN {X 0,Y 295.527,Z 517.21,A -85,B 0,C 180,E1 -18149.349,E2 -18149.349} C_VEL
LIN {X 0,Y 292.679,Z 529.075,A -85,B 0,C 180,E1 -18150.393,E2 -18150.393} C_VEL
LIN {X 0,Y 289.331,Z 540.984,A -85,B 0,C 180,E1 -18151.728,E2 -18151.728} C_VEL
LIN {X 0,Y 285.582,Z 552.247,A -85,B 0,C 180,E1 -18153.313,E2 -18153.313} C_VEL
LIN {X 0,Y 282.153,Z 561.536,A -85,B 0,C 180,E1 -18154.948,E2 -18154.948} C_VEL
LIN {X 0,Y 278.983,Z 569.342,A -85,B 0,C 180,E1 -18156.624,E2 -18156.624} C_VEL
LIN {X 0,Y 275.488,Z 577.092,A -85,B 0,C 180,E1 -18158.683,E2 -18158.683} C_VEL
LIN {X 0,Y 272.922,Z 582.433,A -85,B 0,C 180,E1 -18160.442,E2 -18160.442} C_VEL
LIN {X 0,Y 270.137,Z 587.679,A -85,B 0,C 180,E1 -18162.591,E2 -18162.591} C_VEL
LIN {X 0,Y 267.803,Z 591.779,A -85,B 0,C 180,E1 -18164.786,E2 -18164.786} C_VEL
LIN {X 0,Y 266.333,Z 593.936,A -85,B 0,C 180,E1 -18166.262,E2 -18166.262} C_VEL
LIN {X 0,Y 265.233,Z 595.649,A -85,B 0,C 180,E1 -18167.762,E2 -18167.762} C_VEL
LIN {X 0,Y 264.349,Z 596.898,A -85,B 0,C 180,E1 -18169.275,E2 -18169.275} C_VEL
LIN {X 0,Y 263.38,Z 597.787,A -85,B 0,C 180,E1 -18170.87,E2 -18170.87} C_VEL
LIN {X 0,Y 262.155,Z 598.244,A -85,B 0,C 180,E1 -18173.844,E2 -18173.844} C_VEL
LIN {X 0,Y 261.806,Z 597.826,A -85,B 0,C 180,E1 -18175.381,E2 -18175.381} C_VEL
LIN {X 0,Y 261.545,Z 597.003,A -85,B 0,C 180,E1 -18176.919,E2 -18176.919} C_VEL
LIN {X 0,Y 261.333,Z 595.776,A -85,B 0,C 180,E1 -18178.459,E2 -18178.459} C_VEL
LIN {X 0,Y 261.199,Z 593.08,A -85,B 0,C 180,E1 -18180.771,E2 -18180.771} C_VEL
LIN {X 0,Y 261.317,Z 589.334,A -85,B 0,C 180,E1 -18183.084,E2 -18183.084} C_VEL
LIN {X 0,Y 261.354,Z 584.854,A -85,B 0,C 180,E1 -18185.203,E2 -18185.203} C_VEL
LIN {X 0,Y 261.766,Z 578.118,A -85,B 0,C 180,E1 -18187.715,E2 -18187.715} C_VEL
LIN {X 0,Y 262.249,Z 570.305,A -85,B 0,C 180,E1 -18190.032,E2 -18190.032} C_VEL
LIN {X 0,Y 262.863,Z 562.358,A -85,B 0,C 180,E1 -18191.959,E2 -18191.959} C_VEL
LIN {X 0,Y 263.757,Z 551.654,A -85,B 0,C 180,E1 -18194.072,E2 -18194.072} C_VEL
LIN {X 0,Y 264.667,Z 540.942,A -85,B 0,C 180,E1 -18195.794,E2 -18195.794} C_VEL
LIN {X 0,Y 265.572,Z 528.749,A -85,B 0,C 180,E1 -18197.362,E2 -18197.362} C_VEL
LIN {X 0,Y 266.392,Z 515.908,A -85,B 0,C 180,E1 -18198.656,E2 -18198.656} C_VEL
LIN {X 0,Y 267.189,Z 502.225,A -85,B 0,C 180,E1 -18199.695,E2 -18199.695} C_VEL
LIN {X 0,Y 267.87,Z 487.956,A -85,B 0,C 180,E1 -18200.443,E2 -18200.443} C_VEL
LIN {X 0,Y 270.847,Z 411.915,A -85,B 0,C 180,E1 -18203.569,E2 -18203.569} C_VEL
LIN {X 0,Y 267.6,Z 385.045,A -85,B 0,C 180,E1 -18204.848,E2 -18204.848} C_VEL
LIN {X 0,Y 267.443,Z 382.745,A -85,B 0,C 180,E1 -18204.96,E2 -18204.96} C_VEL
LIN {X 0,Y 265.062,Z 370.054,A -85,B 0,C 180,E1 -18208.076,E2 -18208.076} C_VEL
LIN {X 0,Y 263.244,Z 361.318,A -85,B 0,C 180,E1 -18210.299,E2 -18210.299} C_VEL
LIN {X 0,Y 263.158,Z 361.328,A -85,B 0,C 180,E1 -18214.114,E2 -18214.114} C_VEL
LIN {X 0,Y 263.11,Z 361.337,A -85,B 0,C 180,E1 -18217.906,E2 -18217.906} C_VEL
LIN {X 0,Y 263.082,Z 361.343,A -85,B 0,C 180,E1 -18221.902,E2 -18221.902} C_VEL
LIN {X 0,Y 263.085,Z 361.342,A -85,B 0,C 180,E1 -18226.16,E2 -18226.16} C_VEL
LIN {X 0,Y 263.142,Z 361.39,A -85,B 0,C 180,E1 -18229.631,E2 -18229.631} C_VEL
LIN {X 0,Y 264.257,Z 365.394,A -85,B 0,C 180,E1 -18231.338,E2 -18231.338} C_VEL
LIN {X 0,Y 272.166,Z 379.572,A -85,B 0,C 180,E1 -18233.122,E2 -18233.122} C_VEL
LIN {X 0,Y 281.393,Z 398.274,A -85,B 0,C 180,E1 -18235.096,E2 -18235.096} C_VEL
LIN {X 0,Y 287.952,Z 414.038,A -85,B 0,C 180,E1 -18236.469,E2 -18236.469} C_VEL
LIN {X 0,Y 285.533,Z 479.044,A -85,B 0,C 180,E1 -18238.055,E2 -18238.055} C_VEL
LIN {X 0,Y 284.452,Z 503.57,A -85,B 0,C 180,E1 -18238.697,E2 -18238.697} C_VEL
LIN {X 0,Y 283.454,Z 516.118,A -85,B 0,C 180,E1 -18239.242,E2 -18239.242} C_VEL
LIN {X 0,Y 281.757,Z 529.684,A -85,B 0,C 180,E1 -18240.073,E2 -18240.073} C_VEL
LIN {X 0,Y 279.956,Z 541.997,A -85,B 0,C 180,E1 -18241.1,E2 -18241.1} C_VEL
LIN {X 0,Y 278.022,Z 553.081,A -85,B 0,C 180,E1 -18242.265,E2 -18242.265} C_VEL
LIN {X 0,Y 275.608,Z 565.419,A -85,B 0,C 180,E1 -18243.902,E2 -18243.902} C_VEL
LIN {X 0,Y 272.992,Z 576.323,A -85,B 0,C 180,E1 -18245.673,E2 -18245.673} C_VEL
LIN {X 0,Y 270.377,Z 587.079,A -85,B 0,C 180,E1 -18247.856,E2 -18247.856} C_VEL
LIN {X 0,Y 267.982,Z 595.958,A -85,B 0,C 180,E1 -18250.064,E2 -18250.064} C_VEL
LIN {X 0,Y 265.853,Z 604.454,A -85,B 0,C 180,E1 -18252.696,E2 -18252.696} C_VEL
LIN {X 0,Y 264.61,Z 609.497,A -85,B 0,C 180,E1 -18254.595,E2 -18254.595} C_VEL
LIN {X 0,Y 263.226,Z 614.586,A -85,B 0,C 180,E1 -18256.88,E2 -18256.88} C_VEL
LIN {X 0,Y 262.332,Z 618.664,A -85,B 0,C 180,E1 -18259.189,E2 -18259.189} C_VEL
LIN {X 0,Y 261.56,Z 622.792,A -85,B 0,C 180,E1 -18262.277,E2 -18262.277} C_VEL
LIN {X 0,Y 261.145,Z 625.495,A -85,B 0,C 180,E1 -18265.367,E2 -18265.367} C_VEL
LIN {X 0,Y 261.053,Z 626.849,A -85,B 0,C 180,E1 -18268.455,E2 -18268.455} C_VEL
LIN {X 0,Y 261.075,Z 627.029,A -85,B 0,C 180,E1 -18269.998,E2 -18269.998} C_VEL
LIN {X 0,Y 261.08,Z 626.401,A -85,B 0,C 180,E1 -18273.084,E2 -18273.084} C_VEL
LIN {X 0,Y 261.317,Z 624.437,A -85,B 0,C 180,E1 -18276.173,E2 -18276.173} C_VEL
LIN {X 0,Y 261.86,Z 621.088,A -85,B 0,C 180,E1 -18279.264,E2 -18279.264} C_VEL
LIN {X 0,Y 262.898,Z 616.253,A -85,B 0,C 180,E1 -18282.346,E2 -18282.346} C_VEL
LIN {X 0,Y 264.066,Z 611.591,A -85,B 0,C 180,E1 -18284.643,E2 -18284.643} C_VEL
LIN {X 0,Y 265.512,Z 605.879,A -85,B 0,C 180,E1 -18286.925,E2 -18286.925} C_VEL
LIN {X 0,Y 267.606,Z 597.739,A -85,B 0,C 180,E1 -18289.561,E2 -18289.561} C_VEL
LIN {X 0,Y 269.882,Z 589.219,A -85,B 0,C 180,E1 -18291.78,E2 -18291.78} C_VEL
LIN {X 0,Y 272.476,Z 578.892,A -85,B 0,C 180,E1 -18293.966,E2 -18293.966} C_VEL
LIN {X 0,Y 275.234,Z 567.338,A -85,B 0,C 180,E1 -18295.928,E2 -18295.928} C_VEL
LIN {X 0,Y 277.713,Z 555.17,A -85,B 0,C 180,E1 -18297.594,E2 -18297.594} C_VEL
LIN {X 0,Y 279.802,Z 543.116,A -85,B 0,C 180,E1 -18298.912,E2 -18298.912} C_VEL
LIN {X 0,Y 281.834,Z 529.973,A -85,B 0,C 180,E1 -18300.016,E2 -18300.016} C_VEL
LIN {X 0,Y 283.525,Z 515.75,A -85,B 0,C 180,E1 -18300.899,E2 -18300.899} C_VEL
LIN {X 0,Y 284.635,Z 502.029,A -85,B 0,C 180,E1 -18301.476,E2 -18301.476} C_VEL
LIN {X 0,Y 286.716,Z 450.42,A -85,B 0,C 180,E1 -18302.755,E2 -18302.755} C_VEL
LIN {X 0,Y 288.062,Z 414.274,A -85,B 0,C 180,E1 -18303.637,E2 -18303.637} C_VEL
LIN {X 0,Y 281.228,Z 398.004,A -85,B 0,C 180,E1 -18305.066,E2 -18305.066} C_VEL
LIN {X 0,Y 273.17,Z 381.457,A -85,B 0,C 180,E1 -18306.793,E2 -18306.793} C_VEL
LIN {X 0,Y 266.338,Z 369.148,A -85,B 0,C 180,E1 -18308.316,E2 -18308.316} C_VEL
LIN {X 0,Y 264.153,Z 365.144,A -85,B 0,C 180,E1 -18308.875,E2 -18308.875} C_VEL
LIN {X 0,Y 263.08,Z 361.338,A -85,B 0,C 180,E1 -18310.544,E2 -18310.544} C_VEL
LIN {X 0,Y 263.068,Z 361.34,A -85,B 0,C 180,E1 -18313.992,E2 -18313.992} C_VEL
LIN {X 0,Y 263.044,Z 361.339,A -85,B 0,C 180,E1 -18316.595,E2 -18316.595} C_VEL
LIN {X 0,Y 262.362,Z 361.429,A -85,B 0,C 180,E1 -18317.874,E2 -18317.874} C_VEL
LIN {X 0,Y 259.564,Z 361.778,A -85,B 0,C 180,E1 -18319.96,E2 -18319.96} C_VEL
LIN {X 0,Y 257.191,Z 362.065,A -85,B 0,C 180,E1 -18321.656,E2 -18321.656} C_VEL
LIN {X 0,Y 256.152,Z 362.19,A -85,B 0,C 180,E1 -18322.97,E2 -18322.97} C_VEL
LIN {X 0,Y 256.055,Z 362.201,A -85,B 0,C 180,E1 -18323.415,E2 -18323.415} C_VEL
LIN {X 0,Y 256.055,Z 362.195,A -85,B 0,C 180,E1 -18326.705,E2 -18326.705} C_VEL
LIN {X 0,Y 256.044,Z 362.217,A -85,B 0,C 180,E1 -18330.391,E2 -18330.391} C_VEL
LIN {X 0,Y 256.121,Z 362.187,A -85,B 0,C 180,E1 -18334.887,E2 -18334.887} C_VEL
LIN {X 0,Y 256.111,Z 362.19,A -85,B 0,C 180,E1 -18339.1,E2 -18339.1} C_VEL
LIN {X 0,Y 256.218,Z 362.192,A -85,B 0,C 180,E1 -18344.08,E2 -18344.08} C_VEL
LIN {X 0,Y 256.277,Z 362.188,A -85,B 0,C 180,E1 -18348.932,E2 -18348.932} C_VEL
LIN {X 0,Y 256.454,Z 362.16,A -85,B 0,C 180,E1 -18352.124,E2 -18352.124} C_VEL
LIN {X 0,Y 256.441,Z 362.165,A -85,B 0,C 180,E1 -18356.858,E2 -18356.858} C_VEL
LIN {X 0,Y 256.683,Z 362.134,A -85,B 0,C 180,E1 -18358.431,E2 -18358.431} C_VEL
LIN {X 0,Y 256.687,Z 362.135,A -85,B 0,C 180,E1 -18361.569,E2 -18361.569} C_VEL
LIN {X 0,Y 256.441,Z 362.167,A -85,B 0,C 180,E1 -18366.294,E2 -18366.294} C_VEL
LIN {X 0,Y 256.414,Z 362.166,A -85,B 0,C 180,E1 -18369.465,E2 -18369.465} C_VEL
LIN {X 0,Y 256.218,Z 362.192,A -85,B 0,C 180,E1 -18374.292,E2 -18374.292} C_VEL
LIN {X 0,Y 256.15,Z 362.198,A -85,B 0,C 180,E1 -18377.566,E2 -18377.566} C_VEL
LIN {X 0,Y 256.106,Z 362.187,A -85,B 0,C 180,E1 -18381.098,E2 -18381.098} C_VEL
LIN {X 0,Y 256.069,Z 362.212,A -85,B 0,C 180,E1 -18385.088,E2 -18385.088} C_VEL
LIN {X 0,Y 256.064,Z 362.191,A -85,B 0,C 180,E1 -18388.57,E2 -18388.57} C_VEL
LIN {X 0,Y 256.058,Z 362.214,A -85,B 0,C 180,E1 -18391.701,E2 -18391.701} C_VEL
LIN {X 0,Y 256.068,Z 362.213,A -85,B 0,C 180,E1 -18395.195,E2 -18395.195} C_VEL
LIN {X 0,Y 256.054,Z 362.213,A -85,B 0,C 180,E1 -18399.145,E2 -18399.145} C_VEL
LIN {X 0,Y 256.012,Z 362.219,A -85,B 0,C 180,E1 -18403.338,E2 -18403.338} C_VEL
LIN {X 0,Y 256.029,Z 362.322,A -85,B 0,C 180,E1 -18407.127,E2 -18407.127} C_VEL
LIN {X 0,Y 258.044,Z 369.065,A -85,B 0,C 180,E1 -18410.12,E2 -18410.12} C_VEL
LIN {X 0,Y 265.843,Z 383.294,A -85,B 0,C 180,E1 -18411.988,E2 -18411.988} C_VEL
LIN {X 0,Y 272.629,Z 396.832,A -85,B 0,C 180,E1 -18413.528,E2 -18413.528} C_VEL
LIN {X 0,Y 280.309,Z 414.562,A -85,B 0,C 180,E1 -18415.221,E2 -18415.221} C_VEL
LIN {X 0,Y 281.532,Z 418.47,A -85,B 0,C 180,E1 -18415.512,E2 -18415.512} C_VEL
LIN {X 0,Y 281.947,Z 422.437,A -85,B 0,C 180,E1 -18415.69,E2 -18415.69} C_VEL
LIN {X 0,Y 279.008,Z 495.186,A -85,B 0,C 180,E1 -18417.479,E2 -18417.479} C_VEL
LIN {X 0,Y 278.192,Z 511.008,A -85,B 0,C 180,E1 -18417.962,E2 -18417.962} C_VEL
LIN {X 0,Y 276.739,Z 524.971,A -85,B 0,C 180,E1 -18418.63,E2 -18418.63} C_VEL
LIN {X 0,Y 274.879,Z 538.562,A -85,B 0,C 180,E1 -18419.568,E2 -18419.568} C_VEL
LIN {X 0,Y 272.781,Z 550.842,A -85,B 0,C 180,E1 -18420.694,E2 -18420.694} C_VEL
LIN {X 0,Y 270.445,Z 562.933,A -85,B 0,C 180,E1 -18422.114,E2 -18422.114} C_VEL
LIN {X 0,Y 267.703,Z 575.133,A -85,B 0,C 180,E1 -18423.916,E2 -18423.916} C_VEL
LIN {X 0,Y 265.113,Z 585.213,A -85,B 0,C 180,E1 -18425.742,E2 -18425.742} C_VEL
LIN {X 0,Y 262.46,Z 595.235,A -85,B 0,C 180,E1 -18427.986,E2 -18427.986} C_VEL
LIN {X 0,Y 260.13,Z 603.558,A -85,B 0,C 180,E1 -18430.265,E2 -18430.265} C_VEL
LIN {X 0,Y 258.118,Z 611.518,A -85,B 0,C 180,E1 -18432.983,E2 -18432.983} C_VEL
LIN {X 0,Y 256.418,Z 617.924,A -85,B 0,C 180,E1 -18435.722,E2 -18435.722} C_VEL
LIN {X 0,Y 255.042,Z 623.606,A -85,B 0,C 180,E1 -18438.881,E2 -18438.881} C_VEL
LIN {X 0,Y 254.298,Z 627.732,A -85,B 0,C 180,E1 -18442.06,E2 -18442.06} C_VEL
LIN {X 0,Y 253.972,Z 630.421,A -85,B 0,C 180,E1 -18445.24,E2 -18445.24} C_VEL
LIN {X 0,Y 253.943,Z 631.748,A -85,B 0,C 180,E1 -18448.417,E2 -18448.417} C_VEL
LIN {X 0,Y 253.98,Z 631.911,A -85,B 0,C 180,E1 -18450.002,E2 -18450.002} C_VEL
LIN {X 0,Y 253.912,Z 631.233,A -85,B 0,C 180,E1 -18453.176,E2 -18453.176} C_VEL
LIN {X 0,Y 254.076,Z 629.211,A -85,B 0,C 180,E1 -18456.355,E2 -18456.355} C_VEL
LIN {X 0,Y 254.634,Z 625.802,A -85,B 0,C 180,E1 -18459.535,E2 -18459.535} C_VEL
LIN {X 0,Y 255.588,Z 620.902,A -85,B 0,C 180,E1 -18462.71,E2 -18462.71} C_VEL
LIN {X 0,Y 256.887,Z 616.174,A -85,B 0,C 180,E1 -18465.067,E2 -18465.067} C_VEL
LIN {X 0,Y 258.674,Z 609.266,A -85,B 0,C 180,E1 -18467.819,E2 -18467.819} C_VEL
LIN {X 0,Y 260.133,Z 603.555,A -85,B 0,C 180,E1 -18469.74,E2 -18469.74} C_VEL
LIN {X 0,Y 263.212,Z 596.379,A -85,B 0,C 180,E1 -18472.366,E2 -18472.366} C_VEL
LIN {X 0,Y 266.859,Z 587.515,A -85,B 0,C 180,E1 -18474.924,E2 -18474.924} C_VEL
LIN {X 0,Y 270.613,Z 578.211,A -85,B 0,C 180,E1 -18477.034,E2 -18477.034} C_VEL
LIN {X 0,Y 274.792,Z 567.01,A -85,B 0,C 180,E1 -18479.076,E2 -18479.076} C_VEL
LIN {X 0,Y 278.542,Z 555.794,A -85,B 0,C 180,E1 -18480.728,E2 -18480.728} C_VEL
LIN {X 0,Y 281.955,Z 544.965,A -85,B 0,C 180,E1 -18481.986,E2 -18481.986} C_VEL
LIN {X 0,Y 285.54,Z 531.976,A -85,B 0,C 180,E1 -18483.176,E2 -18483.176} C_VEL
LIN {X 0,Y 288.905,Z 517.336,A -85,B 0,C 180,E1 -18484.182,E2 -18484.182} C_VEL
LIN {X 0,Y 294.649,Z 485.61,A -85,B 0,C 180,E1 -18485.656,E2 -18485.656} C_VEL
LIN {X 0,Y 304.778,Z 431.033,A -85,B 0,C 180,E1 -18488.115,E2 -18488.115} C_VEL
LIN {X 0,Y 304.249,Z 429.802,A -85,B 0,C 180,E1 -18488.654,E2 -18488.654} C_VEL
LIN {X 0,Y 302.449,Z 426.903,A -85,B 0,C 180,E1 -18490.592,E2 -18490.592} C_VEL
LIN {X 0,Y 301.277,Z 425.33,A -85,B 0,C 180,E1 -18492.365,E2 -18492.365} C_VEL
LIN {X 0,Y 300.479,Z 424.732,A -85,B 0,C 180,E1 -18494.564,E2 -18494.564} C_VEL
LIN {X 0,Y 300.52,Z 425.157,A -85,B 0,C 180,E1 -18496.878,E2 -18496.878} C_VEL
LIN {X 0,Y 301.03,Z 426.555,A -85,B 0,C 180,E1 -18498.566,E2 -18498.566} C_VEL
LIN {X 0,Y 302.342,Z 429.727,A -85,B 0,C 180,E1 -18500.804,E2 -18500.804} C_VEL
LIN {X 0,Y 303.971,Z 434.018,A -85,B 0,C 180,E1 -18502.72,E2 -18502.72} C_VEL
LIN {X 0,Y 305.691,Z 439.219,A -85,B 0,C 180,E1 -18504.354,E2 -18504.354} C_VEL
LIN {X 0,Y 294.677,Z 503.505,A -85,B 0,C 180,E1 -18507.242,E2 -18507.242} C_VEL
LIN {X 0,Y 291.645,Z 517.821,A -85,B 0,C 180,E1 -18508.188,E2 -18508.188} C_VEL
LIN {X 0,Y 288.147,Z 531.18,A -85,B 0,C 180,E1 -18509.393,E2 -18509.393} C_VEL
LIN {X 0,Y 284.823,Z 541.995,A -85,B 0,C 180,E1 -18510.632,E2 -18510.632} C_VEL
LIN {X 0,Y 280.491,Z 554.05,A -85,B 0,C 180,E1 -18512.384,E2 -18512.384} C_VEL
LIN {X 0,Y 276.858,Z 563.073,A -85,B 0,C 180,E1 -18514.031,E2 -18514.031} C_VEL
LIN {X 0,Y 272.827,Z 571.986,A -85,B 0,C 180,E1 -18516.064,E2 -18516.064} C_VEL
LIN {X 0,Y 269.167,Z 579.314,A -85,B 0,C 180,E1 -18518.157,E2 -18518.157} C_VEL
LIN {X 0,Y 266.483,Z 584.317,A -85,B 0,C 180,E1 -18519.949,E2 -18519.949} C_VEL
LIN {X 0,Y 263.535,Z 589.253,A -85,B 0,C 180,E1 -18522.141,E2 -18522.141} C_VEL
LIN {X 0,Y 261.073,Z 593.068,A -85,B 0,C 180,E1 -18524.384,E2 -18524.384} C_VEL
LIN {X 0,Y 259.547,Z 595.069,A -85,B 0,C 180,E1 -18525.895,E2 -18525.895} C_VEL
LIN {X 0,Y 257.409,Z 597.679,A -85,B 0,C 180,E1 -18528.982,E2 -18528.982} C_VEL
LIN {X 0,Y 256.364,Z 598.472,A -85,B 0,C 180,E1 -18530.729,E2 -18530.729} C_VEL
LIN {X 0,Y 255.116,Z 598.564,A -85,B 0,C 180,E1 -18533.674,E2 -18533.674} C_VEL
LIN {X 0,Y 254.737,Z 598.028,A -85,B 0,C 180,E1 -18535.252,E2 -18535.252} C_VEL
LIN {X 0,Y 254.48,Z 597.091,A -85,B 0,C 180,E1 -18536.834,E2 -18536.834} C_VEL
LIN {X 0,Y 254.259,Z 595.689,A -85,B 0,C 180,E1 -18538.416,E2 -18538.416} C_VEL
LIN {X 0,Y 254.126,Z 592.783,A -85,B 0,C 180,E1 -18540.792,E2 -18540.792} C_VEL
LIN {X 0,Y 254.253,Z 588.802,A -85,B 0,C 180,E1 -18543.169,E2 -18543.169} C_VEL
LIN {X 0,Y 254.367,Z 582.732,A -85,B 0,C 180,E1 -18545.91,E2 -18545.91} C_VEL
LIN {X 0,Y 254.772,Z 575.849,A -85,B 0,C 180,E1 -18548.327,E2 -18548.327} C_VEL
LIN {X 0,Y 255.337,Z 567.379,A -85,B 0,C 180,E1 -18550.707,E2 -18550.707} C_VEL
LIN {X 0,Y 256.005,Z 558.787,A -85,B 0,C 180,E1 -18552.687,E2 -18552.687} C_VEL
LIN {X 0,Y 257.031,Z 547.17,A -85,B 0,C 180,E1 -18554.853,E2 -18554.853} C_VEL
LIN {X 0,Y 257.968,Z 535.252,A -85,B 0,C 180,E1 -18556.622,E2 -18556.622} C_VEL
LIN {X 0,Y 258.87,Z 522.904,A -85,B 0,C 180,E1 -18558.081,E2 -18558.081} C_VEL
LIN {X 0,Y 259.81,Z 508.789,A -85,B 0,C 180,E1 -18559.352,E2 -18559.352} C_VEL
LIN {X 0,Y 260.438,Z 495.464,A -85,B 0,C 180,E1 -18560.228,E2 -18560.228} C_VEL
LIN {X 0,Y 262.301,Z 448.398,A -85,B 0,C 180,E1 -18562.29,E2 -18562.29} C_VEL
LIN {X 0,Y 263.792,Z 412.011,A -85,B 0,C 180,E1 -18563.839,E2 -18563.839} C_VEL
LIN {X 0,Y 260.673,Z 385.812,A -85,B 0,C 180,E1 -18565.122,E2 -18565.122} C_VEL
LIN {X 0,Y 260.338,Z 382.896,A -85,B 0,C 180,E1 -18565.303,E2 -18565.303} C_VEL
LIN {X 0,Y 257.374,Z 367.768,A -85,B 0,C 180,E1 -18569.092,E2 -18569.092} C_VEL
LIN {X 0,Y 256.18,Z 362.196,A -85,B 0,C 180,E1 -18570.556,E2 -18570.556} C_VEL
LIN {X 0,Y 256.084,Z 362.212,A -85,B 0,C 180,E1 -18575.193,E2 -18575.193} C_VEL
LIN {X 0,Y 256.048,Z 362.215,A -85,B 0,C 180,E1 -18579.147,E2 -18579.147} C_VEL
LIN {X 0,Y 256.028,Z 362.218,A -85,B 0,C 180,E1 -18583.335,E2 -18583.335} C_VEL
LIN {X 0,Y 256.062,Z 362.217,A -85,B 0,C 180,E1 -18587.822,E2 -18587.822} C_VEL
LIN {X 0,Y 256.059,Z 362.254,A -85,B 0,C 180,E1 -18588.59,E2 -18588.59} C_VEL
LIN {X 0,Y 256.981,Z 365.5,A -85,B 0,C 180,E1 -18590.027,E2 -18590.027} C_VEL
LIN {X 0,Y 265.626,Z 380.616,A -85,B 0,C 180,E1 -18592.088,E2 -18592.088} C_VEL
LIN {X 0,Y 274.001,Z 397.283,A -85,B 0,C 180,E1 -18593.976,E2 -18593.976} C_VEL
LIN {X 0,Y 280.625,Z 412.556,A -85,B 0,C 180,E1 -18595.423,E2 -18595.423} C_VEL
LIN {X 0,Y 282.049,Z 416.178,A -85,B 0,C 180,E1 -18595.732,E2 -18595.732} C_VEL
LIN {X 0,Y 278.636,Z 501.702,A -85,B 0,C 180,E1 -18597.879,E2 -18597.879} C_VEL
LIN {X 0,Y 277.514,Z 514.573,A -85,B 0,C 180,E1 -18598.403,E2 -18598.403} C_VEL
LIN {X 0,Y 275.817,Z 528.63,A -85,B 0,C 180,E1 -18599.254,E2 -18599.254} C_VEL
LIN {X 0,Y 273.767,Z 542.071,A -85,B 0,C 180,E1 -18600.382,E2 -18600.382} C_VEL
LIN {X 0,Y 271.639,Z 553.773,A -85,B 0,C 180,E1 -18601.646,E2 -18601.646} C_VEL
LIN {X 0,Y 269.231,Z 565.491,A -85,B 0,C 180,E1 -18603.235,E2 -18603.235} C_VEL
LIN {X 0,Y 266.535,Z 576.394,A -85,B 0,C 180,E1 -18605.044,E2 -18605.044} C_VEL
LIN {X 0,Y 263.773,Z 587.15,A -85,B 0,C 180,E1 -18607.271,E2 -18607.271} C_VEL
LIN {X 0,Y 261.287,Z 596.027,A -85,B 0,C 180,E1 -18609.531,E2 -18609.531} C_VEL
LIN {X 0,Y 259.137,Z 604.177,A -85,B 0,C 180,E1 -18612.106,E2 -18612.106} C_VEL
LIN {X 0,Y 257.76,Z 609.565,A -85,B 0,C 180,E1 -18614.175,E2 -18614.175} C_VEL
LIN {X 0,Y 256.283,Z 614.655,A -85,B 0,C 180,E1 -18616.518,E2 -18616.518} C_VEL
LIN {X 0,Y 255.072,Z 619.922,A -85,B 0,C 180,E1 -18619.681,E2 -18619.681} C_VEL
LIN {X 0,Y 254.506,Z 622.86,A -85,B 0,C 180,E1 -18622.061,E2 -18622.061} C_VEL
LIN {X 0,Y 254.064,Z 625.563,A -85,B 0,C 180,E1 -18625.237,E2 -18625.237} C_VEL
LIN {X 0,Y 253.964,Z 626.916,A -85,B 0,C 180,E1 -18628.412,E2 -18628.412} C_VEL
LIN {X 0,Y 253.983,Z 627.097,A -85,B 0,C 180,E1 -18629.998,E2 -18629.998} C_VEL
LIN {X 0,Y 253.982,Z 626.468,A -85,B 0,C 180,E1 -18633.17,E2 -18633.17} C_VEL
LIN {X 0,Y 254.246,Z 624.504,A -85,B 0,C 180,E1 -18636.346,E2 -18636.346} C_VEL
LIN {X 0,Y 254.825,Z 621.155,A -85,B 0,C 180,E1 -18639.522,E2 -18639.522} C_VEL
LIN {X 0,Y 255.915,Z 616.32,A -85,B 0,C 180,E1 -18642.689,E2 -18642.689} C_VEL
LIN {X 0,Y 257.192,Z 611.657,A -85,B 0,C 180,E1 -18645.043,E2 -18645.043} C_VEL
LIN {X 0,Y 258.672,Z 605.945,A -85,B 0,C 180,E1 -18647.387,E2 -18647.387} C_VEL
LIN {X 0,Y 260.878,Z 597.804,A -85,B 0,C 180,E1 -18650.086,E2 -18650.086} C_VEL
LIN {X 0,Y 263.283,Z 589.284,A -85,B 0,C 180,E1 -18652.355,E2 -18652.355} C_VEL
LIN {X 0,Y 265.982,Z 578.956,A -85,B 0,C 180,E1 -18654.59,E2 -18654.59} C_VEL
LIN {X 0,Y 268.869,Z 567.401,A -85,B 0,C 180,E1 -18656.589,E2 -18656.589} C_VEL
LIN {X 0,Y 271.486,Z 554.864,A -85,B 0,C 180,E1 -18658.337,E2 -18658.337} C_VEL
LIN {X 0,Y 273.622,Z 543.177,A -85,B 0,C 180,E1 -18659.63,E2 -18659.63} C_VEL
LIN {X 0,Y 275.717,Z 530.033,A -85,B 0,C 180,E1 -18660.754,E2 -18660.754} C_VEL
LIN {X 0,Y 277.477,Z 515.807,A -85,B 0,C 180,E1 -18661.65,E2 -18661.65} C_VEL
LIN {X 0,Y 278.703,Z 501.045,A -85,B 0,C 180,E1 -18662.265,E2 -18662.265} C_VEL
LIN {X 0,Y 281.387,Z 435.087,A -85,B 0,C 180,E1 -18663.918,E2 -18663.918} C_VEL
LIN {X 0,Y 282.114,Z 416.097,A -85,B 0,C 180,E1 -18664.39,E2 -18664.39} C_VEL
LIN {X 0,Y 274.875,Z 399.076,A -85,B 0,C 180,E1 -18665.968,E2 -18665.968} C_VEL
LIN {X 0,Y 266.227,Z 381.706,A -85,B 0,C 180,E1 -18667.913,E2 -18667.913} C_VEL
LIN {X 0,Y 261.471,Z 373.316,A -85,B 0,C 180,E1 -18669.02,E2 -18669.02} C_VEL
LIN {X 0,Y 258.521,Z 368.499,A -85,B 0,C 180,E1 -18669.723,E2 -18669.723} C_VEL
LIN {X 0,Y 256.853,Z 365.256,A -85,B 0,C 180,E1 -18670.188,E2 -18670.188} C_VEL
LIN {X 0,Y 256.02,Z 362.219,A -85,B 0,C 180,E1 -18671.617,E2 -18671.617} C_VEL
LIN {X 0,Y 256.009,Z 362.221,A -85,B 0,C 180,E1 -18675.537,E2 -18675.537} C_VEL
LIN {X 0,Y 256.009,Z 362.218,A -85,B 0,C 180,E1 -18678.787,E2 -18678.787} C_VEL
LIN {X 0,Y 256.092,Z 362.196,A -85,B 0,C 180,E1 -18682.861,E2 -18682.861} C_VEL
LIN {X 0,Y 256.055,Z 362.201,A -85,B 0,C 180,E1 -18683.415,E2 -18683.415} C_VEL
LIN {X 0,Y 255.346,Z 362.304,A -85,B 0,C 180,E1 -18684.728,E2 -18684.728} C_VEL
LIN {X 0,Y 252.463,Z 362.655,A -85,B 0,C 180,E1 -18686.87,E2 -18686.87} C_VEL
LIN {X 0,Y 250.057,Z 362.954,A -85,B 0,C 180,E1 -18688.612,E2 -18688.612} C_VEL
LIN {X 0,Y 249.056,Z 363.086,A -85,B 0,C 180,E1 -18689.964,E2 -18689.964} C_VEL
LIN {X 0,Y 248.99,Z 363.089,A -85,B 0,C 180,E1 -18690.422,E2 -18690.422} C_VEL
LIN {X 0,Y 249.09,Z 363.063,A -85,B 0,C 180,E1 -18694.962,E2 -18694.962} C_VEL
LIN {X 0,Y 249.042,Z 363.076,A -85,B 0,C 180,E1 -18698.625,E2 -18698.625} C_VEL
LIN {X 0,Y 249.145,Z 363.072,A -85,B 0,C 180,E1 -18703.615,E2 -18703.615} C_VEL
LIN {X 0,Y 249.22,Z 363.067,A -85,B 0,C 180,E1 -18708.615,E2 -18708.615} C_VEL
LIN {X 0,Y 249.404,Z 363.038,A -85,B 0,C 180,E1 -18711.9,E2 -18711.9} C_VEL
LIN {X 0,Y 249.251,Z 363.052,A -85,B 0,C 180,E1 -18715.147,E2 -18715.147} C_VEL
LIN {X 0,Y 249.644,Z 363.011,A -85,B 0,C 180,E1 -18718.387,E2 -18718.387} C_VEL
LIN {X 0,Y 249.647,Z 363.012,A -85,B 0,C 180,E1 -18721.613,E2 -18721.613} C_VEL
LIN {X 0,Y 249.412,Z 363.044,A -85,B 0,C 180,E1 -18726.472,E2 -18726.472} C_VEL
LIN {X 0,Y 249.33,Z 363.049,A -85,B 0,C 180,E1 -18729.737,E2 -18729.737} C_VEL
LIN {X 0,Y 249.158,Z 363.075,A -85,B 0,C 180,E1 -18734.706,E2 -18734.706} C_VEL
LIN {X 0,Y 249.082,Z 363.08,A -85,B 0,C 180,E1 -18738.082,E2 -18738.082} C_VEL
LIN {X 0,Y 249.03,Z 363.064,A -85,B 0,C 180,E1 -18741.523,E2 -18741.523} C_VEL
LIN {X 0,Y 249.031,Z 363.089,A -85,B 0,C 180,E1 -18745.441,E2 -18745.441} C_VEL
LIN {X 0,Y 249.012,Z 363.068,A -85,B 0,C 180,E1 -18748.969,E2 -18748.969} C_VEL
LIN {X 0,Y 249.014,Z 363.09,A -85,B 0,C 180,E1 -18752.428,E2 -18752.428} C_VEL
LIN {X 0,Y 249.002,Z 363.09,A -85,B 0,C 180,E1 -18756.35,E2 -18756.35} C_VEL
LIN {X 0,Y 248.968,Z 363.097,A -85,B 0,C 180,E1 -18760.485,E2 -18760.485} C_VEL
LIN {X 0,Y 248.952,Z 363.102,A -85,B 0,C 180,E1 -18764.891,E2 -18764.891} C_VEL
LIN {X 0,Y 248.967,Z 363.152,A -85,B 0,C 180,E1 -18765.985,E2 -18765.985} C_VEL
LIN {X 0,Y 250.617,Z 368.928,A -85,B 0,C 180,E1 -18768.684,E2 -18768.684} C_VEL
LIN {X 0,Y 253.14,Z 373.268,A -85,B 0,C 180,E1 -18769.342,E2 -18769.342} C_VEL
LIN {X 0,Y 259.524,Z 384.619,A -85,B 0,C 180,E1 -18770.937,E2 -18770.937} C_VEL
LIN {X 0,Y 266.58,Z 398.538,A -85,B 0,C 180,E1 -18772.619,E2 -18772.619} C_VEL
LIN {X 0,Y 273.897,Z 415.227,A -85,B 0,C 180,E1 -18774.307,E2 -18774.307} C_VEL
LIN {X 0,Y 275.845,Z 420.8,A -85,B 0,C 180,E1 -18774.771,E2 -18774.771} C_VEL
LIN {X 0,Y 276.018,Z 425.13,A -85,B 0,C 180,E1 -18774.931,E2 -18774.931} C_VEL
LIN {X 0,Y 272.542,Z 506.935,A -85,B 0,C 180,E1 -18777.022,E2 -18777.022} C_VEL
LIN {X 0,Y 271.134,Z 521.103,A -85,B 0,C 180,E1 -18777.63,E2 -18777.63} C_VEL
LIN {X 0,Y 269.266,Z 535.112,A -85,B 0,C 180,E1 -18778.536,E2 -18778.536} C_VEL
LIN {X 0,Y 266.936,Z 549.012,A -85,B 0,C 180,E1 -18779.769,E2 -18779.769} C_VEL
LIN {X 0,Y 264.446,Z 561.448,A -85,B 0,C 180,E1 -18781.207,E2 -18781.207} C_VEL
LIN {X 0,Y 261.622,Z 573.982,A -85,B 0,C 180,E1 -18783.046,E2 -18783.046} C_VEL
LIN {X 0,Y 258.634,Z 585.148,A -85,B 0,C 180,E1 -18785.093,E2 -18785.093} C_VEL
LIN {X 0,Y 255.862,Z 595.17,A -85,B 0,C 180,E1 -18787.387,E2 -18787.387} C_VEL
LIN {X 0,Y 253.412,Z 603.492,A -85,B 0,C 180,E1 -18789.719,E2 -18789.719} C_VEL
LIN {X 0,Y 251.309,Z 611.452,A -85,B 0,C 180,E1 -18792.507,E2 -18792.507} C_VEL
LIN {X 0,Y 249.505,Z 617.857,A -85,B 0,C 180,E1 -18795.317,E2 -18795.317} C_VEL
LIN {X 0,Y 248.046,Z 623.539,A -85,B 0,C 180,E1 -18798.563,E2 -18798.563} C_VEL
LIN {X 0,Y 247.247,Z 627.665,A -85,B 0,C 180,E1 -18801.832,E2 -18801.832} C_VEL
LIN {X 0,Y 246.881,Z 630.354,A -85,B 0,C 180,E1 -18805.103,E2 -18805.103} C_VEL
LIN {X 0,Y 246.855,Z 631.681,A -85,B 0,C 180,E1 -18808.371,E2 -18808.371} C_VEL
LIN {X 0,Y 246.89,Z 631.844,A -85,B 0,C 180,E1 -18810.002,E2 -18810.002} C_VEL
LIN {X 0,Y 246.82,Z 631.165,A -85,B 0,C 180,E1 -18813.267,E2 -18813.267} C_VEL
LIN {X 0,Y 247.016,Z 629.143,A -85,B 0,C 180,E1 -18816.537,E2 -18816.537} C_VEL
LIN {X 0,Y 247.6,Z 625.733,A -85,B 0,C 180,E1 -18819.808,E2 -18819.808} C_VEL
LIN {X 0,Y 248.624,Z 620.833,A -85,B 0,C 180,E1 -18823.072,E2 -18823.072} C_VEL
LIN {X 0,Y 249.997,Z 616.105,A -85,B 0,C 180,E1 -18825.492,E2 -18825.492} C_VEL
LIN {X 0,Y 251.887,Z 608.864,A -85,B 0,C 180,E1 -18828.442,E2 -18828.442} C_VEL
LIN {X 0,Y 253.546,Z 604.535,A -85,B 0,C 180,E1 -18830.275,E2 -18830.275} C_VEL
LIN {X 0,Y 256.804,Z 597.829,A -85,B 0,C 180,E1 -18832.956,E2 -18832.956} C_VEL
LIN {X 0,Y 260.68,Z 589.457,A -85,B 0,C 180,E1 -18835.556,E2 -18835.556} C_VEL
LIN {X 0,Y 264.631,Z 580.752,A -85,B 0,C 180,E1 -18837.697,E2 -18837.697} C_VEL
LIN {X 0,Y 269.014,Z 570.286,A -85,B 0,C 180,E1 -18839.763,E2 -18839.763} C_VEL
LIN {X 0,Y 272.74,Z 560.482,A -85,B 0,C 180,E1 -18841.347,E2 -18841.347} C_VEL
LIN {X 0,Y 276.938,Z 548.782,A -85,B 0,C 180,E1 -18842.852,E2 -18842.852} C_VEL
LIN {X 0,Y 281.242,Z 535.047,A -85,B 0,C 180,E1 -18844.214,E2 -18844.214} C_VEL
LIN {X 0,Y 285.107,Z 520.376,A -85,B 0,C 180,E1 -18845.287,E2 -18845.287} C_VEL
LIN {X 0,Y 287.943,Z 507.261,A -85,B 0,C 180,E1 -18845.962,E2 -18845.962} C_VEL
LIN {X 0,Y 296.981,Z 459.911,A -85,B 0,C 180,E1 -18848.129,E2 -18848.129} C_VEL
LIN {X 0,Y 301.781,Z 435.899,A -85,B 0,C 180,E1 -18849.212,E2 -18849.212} C_VEL
LIN {X 0,Y 300.1,Z 433.005,A -85,B 0,C 180,E1 -18851.316,E2 -18851.316} C_VEL
LIN {X 0,Y 299.078,Z 431.846,A -85,B 0,C 180,E1 -18853.242,E2 -18853.242} C_VEL
LIN {X 0,Y 298.62,Z 431.705,A -85,B 0,C 180,E1 -18856.019,E2 -18856.019} C_VEL
LIN {X 0,Y 298.993,Z 432.796,A -85,B 0,C 180,E1 -18857.941,E2 -18857.941} C_VEL
LIN {X 0,Y 300.2,Z 436.258,A -85,B 0,C 180,E1 -18860.465,E2 -18860.465} C_VEL
LIN {X 0,Y 301.678,Z 440.552,A -85,B 0,C 180,E1 -18862.382,E2 -18862.382} C_VEL
LIN {X 0,Y 302.466,Z 443.236,A -85,B 0,C 180,E1 -18863.266,E2 -18863.266} C_VEL
LIN {X 0,Y 291.153,Z 504.971,A -85,B 0,C 180,E1 -18866.068,E2 -18866.068} C_VEL
LIN {X 0,Y 287.734,Z 519.775,A -85,B 0,C 180,E1 -18867.08,E2 -18867.08} C_VEL
LIN {X 0,Y 284.023,Z 532.694,A -85,B 0,C 180,E1 -18868.277,E2 -18868.277} C_VEL
LIN {X 0,Y 280.08,Z 544.38,A -85,B 0,C 180,E1 -18869.669,E2 -18869.669} C_VEL
LIN {X 0,Y 275.519,Z 556.009,A -85,B 0,C 180,E1 -18871.427,E2 -18871.427} C_VEL
LIN {X 0,Y 270.886,Z 566.269,A -85,B 0,C 180,E1 -18873.414,E2 -18873.414} C_VEL
LIN {X 0,Y 266.703,Z 574.659,A -85,B 0,C 180,E1 -18875.479,E2 -18875.479} C_VEL
LIN {X 0,Y 262.262,Z 582.532,A -85,B 0,C 180,E1 -18877.966,E2 -18877.966} C_VEL
LIN {X 0,Y 258.993,Z 587.887,A -85,B 0,C 180,E1 -18880.172,E2 -18880.172} C_VEL
LIN {X 0,Y 256.05,Z 592.122,A -85,B 0,C 180,E1 -18882.427,E2 -18882.427} C_VEL
LIN {X 0,Y 254.353,Z 594.337,A -85,B 0,C 180,E1 -18883.96,E2 -18883.96} C_VEL
LIN {X 0,Y 252.746,Z 596.137,A -85,B 0,C 180,E1 -18885.507,E2 -18885.507} C_VEL
LIN {X 0,Y 251.525,Z 597.503,A -85,B 0,C 180,E1 -18887.083,E2 -18887.083} C_VEL
LIN {X 0,Y 250.487,Z 598.456,A -85,B 0,C 180,E1 -18888.674,E2 -18888.674} C_VEL
LIN {X 0,Y 248.681,Z 599.13,A -85,B 0,C 180,E1 -18891.877,E2 -18891.877} C_VEL
LIN {X 0,Y 248.062,Z 598.874,A -85,B 0,C 180,E1 -18893.493,E2 -18893.493} C_VEL
LIN {X 0,Y 247.671,Z 598.187,A -85,B 0,C 180,E1 -18895.117,E2 -18895.117} C_VEL
LIN {X 0,Y 247.416,Z 597.07,A -85,B 0,C 180,E1 -18896.743,E2 -18896.743} C_VEL
LIN {X 0,Y 247.188,Z 595.547,A -85,B 0,C 180,E1 -18898.371,E2 -18898.371} C_VEL
LIN {X 0,Y 247.054,Z 592.419,A -85,B 0,C 180,E1 -18900.815,E2 -18900.815} C_VEL
LIN {X 0,Y 247.166,Z 588.207,A -85,B 0,C 180,E1 -18903.26,E2 -18903.26} C_VEL
LIN {X 0,Y 247.27,Z 582.45,A -85,B 0,C 180,E1 -18905.839,E2 -18905.839} C_VEL
LIN {X 0,Y 247.681,Z 575.921,A -85,B 0,C 180,E1 -18908.157,E2 -18908.157} C_VEL
LIN {X 0,Y 248.224,Z 567.412,A -85,B 0,C 180,E1 -18910.605,E2 -18910.605} C_VEL
LIN {X 0,Y 248.896,Z 558.767,A -85,B 0,C 180,E1 -18912.641,E2 -18912.641} C_VEL
LIN {X 0,Y 249.925,Z 547.058,A -85,B 0,C 180,E1 -18914.869,E2 -18914.869} C_VEL
LIN {X 0,Y 250.877,Z 535.053,A -85,B 0,C 180,E1 -18916.687,E2 -18916.687} C_VEL
LIN {X 0,Y 251.812,Z 522.55,A -85,B 0,C 180,E1 -18918.194,E2 -18918.194} C_VEL
LIN {X 0,Y 252.763,Z 508.438,A -85,B 0,C 180,E1 -18919.491,E2 -18919.491} C_VEL
LIN {X 0,Y 253.437,Z 493.981,A -85,B 0,C 180,E1 -18920.441,E2 -18920.441} C_VEL
LIN {X 0,Y 256.813,Z 412.864,A -85,B 0,C 180,E1 -18924.075,E2 -18924.075} C_VEL
LIN {X 0,Y 253.72,Z 386.434,A -85,B 0,C 180,E1 -18925.406,E2 -18925.406} C_VEL
LIN {X 0,Y 253.2,Z 383.241,A -85,B 0,C 180,E1 -18925.604,E2 -18925.604} C_VEL
LIN {X 0,Y 250.485,Z 369.462,A -85,B 0,C 180,E1 -18929.109,E2 -18929.109} C_VEL
LIN {X 0,Y 249.111,Z 363.076,A -85,B 0,C 180,E1 -18930.813,E2 -18930.813} C_VEL
LIN {X 0,Y 249.049,Z 363.088,A -85,B 0,C 180,E1 -18935.076,E2 -18935.076} C_VEL
LIN {X 0,Y 249.008,Z 363.091,A -85,B 0,C 180,E1 -18938.384,E2 -18938.384} C_VEL
LIN {X 0,Y 248.974,Z 363.096,A -85,B 0,C 180,E1 -18942.781,E2 -18942.781} C_VEL
LIN {X 0,Y 249.021,Z 363.137,A -85,B 0,C 180,E1 -18947.485,E2 -18947.485} C_VEL
LIN {X 0,Y 249.711,Z 365.618,A -85,B 0,C 180,E1 -18948.614,E2 -18948.614} C_VEL
LIN {X 0,Y 258.258,Z 380.186,A -85,B 0,C 180,E1 -18950.784,E2 -18950.784} C_VEL
LIN {X 0,Y 264.257,Z 391.449,A -85,B 0,C 180,E1 -18952.222,E2 -18952.222} C_VEL
LIN {X 0,Y 271.837,Z 407.594,A -85,B 0,C 180,E1 -18953.973,E2 -18953.973} C_VEL
LIN {X 0,Y 276.083,Z 418.021,A -85,B 0,C 180,E1 -18954.939,E2 -18954.939} C_VEL
LIN {X 0,Y 273.629,Z 478.538,A -85,B 0,C 180,E1 -18956.466,E2 -18956.466} C_VEL
LIN {X 0,Y 272.432,Z 503.813,A -85,B 0,C 180,E1 -18957.151,E2 -18957.151} C_VEL
LIN {X 0,Y 271.37,Z 516.272,A -85,B 0,C 180,E1 -18957.711,E2 -18957.711} C_VEL
LIN {X 0,Y 269.572,Z 529.833,A -85,B 0,C 180,E1 -18958.57,E2 -18958.57} C_VEL
LIN {X 0,Y 267.621,Z 542.144,A -85,B 0,C 180,E1 -18959.632,E2 -18959.632} C_VEL
LIN {X 0,Y 265.461,Z 553.605,A -85,B 0,C 180,E1 -18960.888,E2 -18960.888} C_VEL
LIN {X 0,Y 262.91,Z 565.562,A -85,B 0,C 180,E1 -18962.538,E2 -18962.538} C_VEL
LIN {X 0,Y 260.119,Z 576.465,A -85,B 0,C 180,E1 -18964.385,E2 -18964.385} C_VEL
LIN {X 0,Y 257.675,Z 585.596,A -85,B 0,C 180,E1 -18966.276,E2 -18966.276} C_VEL
LIN {X 0,Y 255.031,Z 594.746,A -85,B 0,C 180,E1 -18968.582,E2 -18968.582} C_VEL
LIN {X 0,Y 252.662,Z 603.208,A -85,B 0,C 180,E1 -18971.239,E2 -18971.239} C_VEL
LIN {X 0,Y 250.924,Z 609.634,A -85,B 0,C 180,E1 -18973.732,E2 -18973.732} C_VEL
LIN {X 0,Y 249.361,Z 614.724,A -85,B 0,C 180,E1 -18976.137,E2 -18976.137} C_VEL
